   //Step 100 On EXIT - Store Identification
   IF #Step100ExitPls THEN
       #VD_Identification := #IO_VIDS.VEMData.Identification;
   END_IF;

   (******************************************************************************)
   (* Step 100 to 300                                                            *)
   (******************************************************************************)

   //Step 100 to 300
   IF #Step100To300Cond THEN
       #StepNbr := 300;
       #Step300EntryPls := TRUE;
   ELSE
       #Step300EntryPls := FALSE;
   END_IF;

   //Step 100 to 300 - Condition
   #Step100To300Cond :=
   #StepNbr = 100 AND
   #IO_VIDS.VEMData.CommandCode = 1001 AND
   #Status > 0 AND
   (#IO_VIDS.IDType = 0 AND #IO_VIDS.VEMData.Identification <> 0 OR #IO_VIDS.IDType > 0 AND #IO_VIDS.VEMData.CarrierID <> 0) AND
   NOT #NewData;

   (******************************************************************************)
   (* Step 200 - Send data                                                       *)
   (******************************************************************************)

   //Step 200 - On Entry - Check VEM data
   #DataValidSnd := #Step200EntryPls AND #IO_VIDS.VEMData.CommandCode <> 0;

   //Step 200 - On Entry - Check VEM data - Error
   IF #Step200EntryPls AND NOT #DataValidSnd THEN
       #Status := #STATUS_MINUS_006;
   END_IF;

   //Step 200 On Entry - VDCommLocalSndDB - Send VEM data TO virtual device
   IF #Step200EntryPls AND #Status > 0 THEN
       #SerializePos := 0;
       #RetVal:=Serialize(SRC_VARIABLE:=#IO_VIDS.VEMData, DEST_ARRAY=>#VEMDataSndArray, POS:=#SerializePos);
       #RetVal:=BLKMOV(SRCBLK := #VEMDataSndArray, DSTBLK => #ptrVEMDataVDCommLocalSnd);
       #RetVal:=BLKMOV(SRCBLK := #IO_VIDS.SpecificDataInit, DSTBLK => #ptrSpecDataVDCommLocalSnd);
       #CmdCodeSent := #IO_VIDS.VEMData.CommandCode;
   END_IF;

   //Step 200 on Active - Step Timer - Start
   #_Step200Tmr(I_StartTimer := #StepNbr = 200,
                I_HoldTimer := FALSE,
                I_MaxTimerValue := 15000,
                O_TimerResult => #Step200TmrElapsed,
                O_TimerValue => #Step200TmrAct);

   //Step 200 On Active - Step Timer - Error overtime
   IF #Step200TmrElapsed THEN
       #Status := #STATUS_MINUS_003;
   END_IF;

   //Step 200 On Active - Step Timer - Memorize maximum
   IF #Step200TmrAct > #Step200TmrActMax THEN
       #Step200TmrActMax := #Step200TmrAct;
   END_IF;

   //Step 200 On Active - Send TO VD
   #SendToVD := #StepNbr = 200 AND #Status>0;

   (******************************************************************************)
   (* Step 200 to 300                                                            *)
   (******************************************************************************)

   //Step 200 to 300
   IF #Step200To300Cond THEN
       #StepNbr := 300;
       #Step200ExitPls := TRUE;
   ELSE
       #Step200ExitPls := FALSE;
   END_IF;

   //Step 200 to 300 - Condition
   #Step200To300Cond := #StepNbr = 200 AND #SendFinished AND #Status > 0;

   (******************************************************************************)
   (* Step 300                                                                   *)
   (******************************************************************************)

   //Step 300 On Entry - VDCommLocalRcvDB - Create pointer TO VEM data
   #ptrVEMDataVDCommLocalRcvStruct.ID := #POINTER_SYNTAX_ID;
   #ptrVEMDataVDCommLocalRcvStruct.DataType := #DATA_TYPE_BYTE;
   #ptrVEMDataVDCommLocalRcvStruct.ReplicationFactor := 256;
   #ptrVEMDataVDCommLocalRcvStruct.DbNbr := UINT_TO_WORD(DB_ANY_TO_UINT(#C_VDCommLocalRcvDB));
   #ptrVEMDataVDCommLocalRcvStruct.CrossAreaPointer := SHL(IN := #VDCOM_VEM_DATA_OFFSET, N := 3) OR #AREA_IDENTIFIER; //Offset 10

   //Step 300 On Entry - VDCommLocalRcvDB - Create pointer TO Specific data
   #ptrSpecDataVDCommLocalRcvStruct.ID := #POINTER_SYNTAX_ID;
   #ptrSpecDataVDCommLocalRcvStruct.DataType := #DATA_TYPE_BYTE;
   #ptrSpecDataVDCommLocalRcvStruct.ReplicationFactor := 2048;
   #ptrSpecDataVDCommLocalRcvStruct.DbNbr := UINT_TO_WORD(DB_ANY_TO_UINT(#C_VDCommLocalRcvDB));
   #ptrSpecDataVDCommLocalRcvStruct.CrossAreaPointer := SHL(IN := #VDCOM_SPEC_DATA_OFFSET, N := 3) OR #AREA_IDENTIFIER; //Offset 10

   //Step 300 On Active - Receive data from virtual device
   IF #StepNbr = 300 AND #NewData THEN

       //Copy received data to VEM data receive structure
       #RetVal := BLKMOV(SRCBLK := #ptrVEMDataVDCommLocalRcv, DSTBLK => #VEMDataRcvArray);
       #DeserializePos := 0;
       #RetVal := Deserialize(SRC_ARRAY := #VEMDataRcvArray, DEST_VARIABLE => #VEMDataRcv, POS := #DeserializePos);

       //Received command code
       #CmdCodeRcvd := #VEMDataRcv.CommandCode;

       //Check error code
       IF #VEMDataRcv.ErrorCode < 0 THEN
           #Status := DINT_TO_INT(#VEMDataRcv.ErrorCode);
           //Data not Valid signal
           #VEMDataNotValid := TRUE;
       ELSE
           //Check data
           #DataValidRcv := NOT #IO_VIDS.GetVEMDataByRFID.Running AND
           #VEMDataRcv.CommandCode = #IO_VIDS.VEMData.CommandCode;

           #DataValidRcvGetVEMDataByRFID := #IO_VIDS.GetVEMDataByRFID.Running AND
           ((#VEMDataRcv.IdType = 0 AND #VEMDataRcv.Identification <> 0) OR (#VEMDataRcv.IdType <> 0 AND #VEMDataRcv.CarrierID <> 0));

           IF #DataValidRcv OR #DataValidRcvGetVEMDataByRFID THEN

               //Status 001 : Success
               #Status := #STATUS_001;

               //Copy all data
               #DeserializePos := 0;
               #RetVal := Deserialize(SRC_ARRAY := #VEMDataRcvArray, DEST_VARIABLE => #IO_VIDS.VEMData, POS := #DeserializePos);
               #RetVal := BLKMOV(SRCBLK := #ptrSpecDataVDCommLocalRcv, DSTBLK => #IO_SpecificData);
               #DeserializePos := 0;
               #RetVal := Deserialize(SRC_ARRAY := #VEMDataRcvArray, DEST_VARIABLE => #IO_VEMData, POS := #DeserializePos);
               #DeserializePos := 0;
               #RetVal := Deserialize(SRC_ARRAY := #VEMDataRcvArray, DEST_VARIABLE => #IO_VEMDataChange, POS := #DeserializePos);

               //Data Valid signal
               #VEMDataValid := TRUE;

           ELSE
               #VEMDataNotValid := TRUE;
               #Status := #STATUS_MINUS_005;
           END_IF;
       END_IF;
   END_IF;

   //Step 300 on Active - Step Timer - Start
   #_Step300Tmr(I_StartTimer := #StepNbr = 300,
                I_HoldTimer := FALSE,
                I_MaxTimerValue := 15000,
                O_TimerResult => #Step300TmrElapsed,
                O_TimerValue => #Step300TmrAct);

   //Step 300 On Active - Step Timer - Error overtime
   IF #Step300TmrElapsed THEN
       #Status := #STATUS_MINUS_009;
   END_IF;

   //Step 300 On Active - Step Timer - Memorize maximum
   IF #Step300TmrAct > #Step300TmrActMax THEN
       #Step300TmrActMax := #Step300TmrAct;
   END_IF;

   (******************************************************************************)
   (* Step 300 to 400                                                            *)
   (******************************************************************************)

   //Step 300 to 400
   IF #Step300To400Cond THEN
       #StepNbr := 400;
       #Step300ExitPls := TRUE;
   ELSE
       #Step300ExitPls := FALSE;
   END_IF;

   //Step 300 TO 400 - Condition
   #Step300To400Cond := #StepNbr = 300 AND #Status = 1;

   (******************************************************************************)
   (* Step XXX to 400                                                            *)
   (******************************************************************************)

   //Step XXX TO 400
   IF #StepNbr > 0 AND #Status < 0 THEN
       #VEMDataNotValid := TRUE;
       #StepNbr := 400;
   END_IF;

   (******************************************************************************)
   (* Step 400 to 0                                                              *)
   (******************************************************************************)

   //Step 400 to 0
   IF #Step400To0Cond THEN
       #StepNbr := 0;
       #Step400ExitPls := TRUE;
   ELSE
       #Step400ExitPls := FALSE;
   END_IF;

   //Step 400 TO 0 - Condition
   #Step400To0Cond := #StepNbr = 400;

   (******************************************************************************)
   (* Step 400 - Finish & Final Status                                           *)
   (******************************************************************************)

   //Step 400 On active - Finish & Final Status
   IF #StepNbr = 400 THEN

       IF #IO_VIDS.GetVEMData.Running THEN
           #IO_VIDS.GetVEMData.Running := FALSE;
           #IO_VIDS.GetVEMData.Status := #Status;
           #IO_VIDS.GetVEMData.Finished := TRUE;
       ELSIF #IO_VIDS.ChangeData.Running THEN
           #IO_VIDS.ChangeData.Running := FALSE;
           #IO_VIDS.ChangeData.Status := #Status;
           #IO_VIDS.ChangeData.Finished := TRUE;
       ELSIF #IO_VIDS.InitTag.Running THEN
           #IO_VIDS.InitTag.Running := FALSE;
           #IO_VIDS.InitTag.Status := #Status;
           #IO_VIDS.InitTag.Finished := TRUE;
       ELSIF #IO_VIDS.GetVEMDataByRFID.Running THEN
           #IO_VIDS.GetVEMDataByRFID.Running := FALSE;
           #IO_VIDS.GetVEMDataByRFID.Status := #Status;
           #IO_VIDS.GetVEMDataByRFID.Finished := TRUE;
       ELSIF #IO_VIDS.ReplaceTag.Running THEN
           #IO_VIDS.ReplaceTag.Running := FALSE;
           #IO_VIDS.ReplaceTag.Status := #Status;
           #IO_VIDS.ReplaceTag.Finished := TRUE;
       ELSIF #IO_VIDS.Track.Running THEN
           #IO_VIDS.Track.Running := FALSE;
           #IO_VIDS.Track.Status := #Status;
           #IO_VIDS.Track.Finished := TRUE;
       ELSIF #IO_VIDS.Confirm.Running THEN
           #IO_VIDS.Confirm.Running := FALSE;
           #IO_VIDS.Confirm.Status := #Status;
           #IO_VIDS.Confirm.Finished := TRUE;
       ELSIF #IO_VIDS.Couple.Running THEN
           #IO_VIDS.Couple.Running := FALSE;
           #IO_VIDS.Couple.Status := #Status;
           #IO_VIDS.Couple.Finished := TRUE;
       ELSIF #IO_VIDS.DeCouple.Running THEN
           #IO_VIDS.DeCouple.Running := FALSE;
           #IO_VIDS.DeCouple.Status := #Status;
           #IO_VIDS.DeCouple.Finished := TRUE;
       ELSIF #IO_VIDS.GetNextID.Running THEN
           #IO_VIDS.GetNextID.Running := FALSE;
           #IO_VIDS.GetNextID.Status := #Status;
           #IO_VIDS.GetNextID.Finished := TRUE;
       ELSIF #IO_VIDS.GetSpecData.Running THEN
           #IO_VIDS.GetSpecData.Running := FALSE;
           #IO_VIDS.GetSpecData.Status := #Status;
           #IO_VIDS.GetSpecData.Finished := TRUE;
       ELSIF #IO_VIDS.PutSpecData.Running THEN
           #IO_VIDS.PutSpecData.Running := FALSE;
           #IO_VIDS.PutSpecData.Status := #Status;
           #IO_VIDS.PutSpecData.Finished := TRUE;
       END_IF;

   ELSE

       #IO_VIDS.GetVEMData.Finished := FALSE;
       #IO_VIDS.ChangeData.Finished := FALSE;
       #IO_VIDS.InitTag.Finished := FALSE;
       #IO_VIDS.GetVEMDataByRFID.Finished := FALSE;
       #IO_VIDS.ReplaceTag.Finished := FALSE;
       #IO_VIDS.Track.Finished := FALSE;
       #IO_VIDS.Confirm.Finished := FALSE;
       #IO_VIDS.Couple.Finished := FALSE;
       #IO_VIDS.DeCouple.Finished := FALSE;
       #IO_VIDS.GetNextID.Finished := FALSE;
       #IO_VIDS.GetSpecData.Finished := FALSE;
       #IO_VIDS.PutSpecData.Finished := FALSE;

   END_IF;

   (******************************************************************************)
   (* CPU1500 - VDComSubSystem                                                   *)
   (******************************************************************************)

   //Reset NewData
   #ResetNewData:=#NewData;

   #MessageLength := DWORD_TO_WORD(#IO_VIDS.VEMData.SpecificDataLength+266);

   #"_LVDComSubSystemS7-1500"(I_CommunicationReset:=#ResetAllRequests,
                              I_SendRequest:=#SendToVD,
                              I_ResetNewData:=#ResetNewData,
                              I_MasterNewMessage:=#IO_VDComm.NewMessageVD,
                              I_MasterSendFinished:=#IO_VDComm.MessageSendDoneVD,
                              I_VDCommRecvDB:=#C_VDCommMasterRcvDB,
                              I_VDCommSendDB:=#C_VDCommMasterSndDB,
                              C_LocalRecvDB:=#C_VDCommLocalRcvDB,
                              C_LocalSendDB:=#C_VDCommLocalSndDB,
                              C_MessType:=20562,
                              C_SubSystem:=#C_SubSystem,
                              C_SendMessLen:=#MessageLength,
                              O_SendFinished=>#SendFinished,
                              O_NewData=>#NewData,
                              IO_MasterSendReq:=#IO_VDComm.MasterSendReq,
                              IO_MasterAckReq:=#IO_VDComm.MasterAckReq,
                              IO_SubSystemDBNr:=#IO_VDComm.VDCommSendDBNr,
                              IO_VDCommSendDB:=#IO_VDComm.VDCommSendDB);


   (******************************************************************************)
   (* Common signals to all submodules                                           *)
   (******************************************************************************)

   //Common signals to all submodules
   #IO_VIDS.PartPres := #PartPres;
   #IO_VIDS.IDType := #C_IDType;
   #IO_VIDS.VEMDataValid := #VEMDataValid;
   #IO_VIDS.VEMDataNotValid := #VEMDataNotValid;
   #IO_VIDS.CmdCodeRcvd := #CmdCodeRcvd;
   #IO_VIDS.CmdCodeSent := #CmdCodeSent;

   (******************************************************************************)
   (* Outputs                                                                    *)
   (******************************************************************************)

   IF #SECTION_OUTPUTS THEN

       #O_GetVEMDataBusy := #BusyGetVEMData;
       #O_Status := #Status;
       #O_Alarm := #Status < 0;
       #O_VEMDataValid := #VEMDataValid;
       #O_VEMDataNotValid := #VEMDataNotValid;

   END_IF;

   (******************************************************************************)
   (* HMI                                                                        *)
   (******************************************************************************)

   IF #SECTION_HMI THEN

       //Decode - BodyType matrix - Car type
       #CarTypeBody := DINT_TO_INT(DWORD_TO_DINT(#IO_VEMData.BodyTypeMatrix) / 100000);

       //Decode - BodyType matrix - Steering
       #SteeringBody := DINT_TO_INT((DWORD_TO_DINT(#IO_VEMData.BodyTypeMatrix) / 100000) MOD 10);

       //Decode - Variant - Car type - First digit
       #CarTypeArray[1] := (CHAR_TO_INT(#IO_VEMData.Variant[1]) - 48) * 100;
       #CarTypeArray[2] := (CHAR_TO_INT(#IO_VEMData.Variant[2]) - 48) * 10;
       #CarTypeArray[3] := (CHAR_TO_INT(#IO_VEMData.Variant[3]) - 48);

       //Decode - Variant - Car type - Summary digits
       #CarTypeVariant := #CarTypeArray[1] + #CarTypeArray[2] + #CarTypeArray[3];

       //Decode - Variant - Steering
       #SteeringVariant := #IO_VEMData.Variant[10];

       //HMI - Message - Part Present - Visible
       IF #IO_VIDS.PartPres THEN
           #H_Master.H_msgPartPresAnim := #VISIBLE;
       ELSE
           #H_Master.H_msgPartPresAnim := #OFF;
       END_IF;

       //HMI - Message - VEM Data Valid - Visible
       IF #VEMDataValid THEN
           #H_Master.H_msgVEMDataValidAnim := #VISIBLE;
       ELSE
           #H_Master.H_msgVEMDataValidAnim := #OFF;
       END_IF;

       //HMI - Message - VEM Data not Valid - Visible
       IF #VEMDataNotValid THEN
           #H_Master.H_msgVEMDataNotValidAnim := #VISIBLE;
       ELSE
           #H_Master.H_msgVEMDataNotValidAnim := #OFF;
       END_IF;

       //HMI - Value - Command code sent
       #H_Master.H_txtCommandCodeSent := #CmdCodeSent;

       //HMI - Value - Command code received
       #H_Master.H_txtCommandCodeRcvd := #CmdCodeRcvd;

       (******************************************************************************)
       (* HMI - Vehicle types                                                        *)
       (******************************************************************************)

       //HMI - Message - Body VEM data
       IF #C_IDType = 0 THEN
           #H_Master.H_msgVEMDataBody := 1;
       ELSE
           #H_Master.H_msgVEMDataBody := 0;
       END_IF;

       //HMI - Message - Carrier VEM data
       IF #C_IDType = 0 THEN
           #H_Master.H_msgVEMDataCarrier := 1;
       ELSE
           #H_Master.H_msgVEMDataCarrier := 0;
       END_IF;

       #H_Master.H_txtIdentification := #IO_VEMData.Identification;                    //HMI - Value - TagID
       #H_Master.H_txtBodyID := #IO_VEMData.BodyID;                                    //HMI - Value - BodyID
       #H_Master.H_txtCarrierID := #IO_VEMData.CarrierID;                              //HMI - Value - CarrierID
       #H_Master.H_txtBodyTypeMatrix := #IO_VEMData.BodyTypeMatrix;                    //HMI - Value - Bodytype matrix
       #H_Master.H_txtRouting := #IO_VEMData.Routing;                                  //HMI - Value - Routing
       #H_Master.H_txtCarrierDestination := #IO_VEMData.Destination;                   //HMI - Value - Carrier Destination
       #H_Master.H_txtWorkUntil := #IO_VEMData.WorkUntil;                              //HMI - Value - Work UNTIL Station
       #H_Master.H_txtWorkAfter := #IO_VEMData.BegWorkAfter;                           //HMI - Value - Start Work After Station
       #H_Master.H_txtBodyCargoStatus := #IO_VEMData.BodyCargoStatus ;                 //HMI - Value - Body Cargo Status
       #H_Master.H_txtCarrierCargoStatus := #IO_VEMData.CarrierCargoStatus;            //HMI - Value - Carrier Cargo Status
       #H_Master.H_txtEquipmentWork := #IO_VEMData.EquipmentWork;                      //HMI - Value - Equipment Work
       #H_Master.H_txtAvailabilityStatus := #IO_VEMData.AvailabilityStatus;            //HMI - Value - Availability Status
       #H_Master.H_txtModelYear := #IO_VEMData.ModelYear;                              //HMI - Value - ModelYear
       #H_Master.H_txtPreSerieInfo := #IO_VEMData.PreSerieInfo;                        //HMI - Value - Preseries Info
       #H_Master.H_txtWorkStatus := #IO_VEMData.WorkStatus;                            //HMI - Value - Work Status
       #H_Master.H_txtBodyType1 := #IO_VEMData.BodyType1;                              //HMI - Value - Bodytype 1
       #H_Master.H_txtBodyType2 := #IO_VEMData.BodyType2;                              //HMI - Value - Bodytype 2
       #H_Master.H_txtRobotProgramNumber := #IO_VEMData.RobotProgramNumber;            //HMI - Value - Robot Program Number
       #H_Master.H_txtPLCProgramNbr := #H_Master.H_txtPLCProgramNbr;                   //HMI - Value - PLC Program Number
       #H_Master.H_txtEquipmentWorkDone := #IO_VEMData.EquipmentWorkDone;              //HMI - Value - Equipment Work Done
       #H_Master.H_txtSequenceNumber := #IO_VEMData.SequenceNumber;                    //HMI - Value - Sequence Number
       #H_Master.H_txtBufferIn := #IO_VEMData.BufferIn;                                //HMI - Value - BufferIn
       #H_Master.H_txtBufferOut := #IO_VEMData.BufferOut;                              //HMI - Value - BufferOut
       #H_Master.H_txtCarrierType := #IO_VEMData.CarrierType;                          //HMI - Value - Carrier Type
       #H_Master.H_txtCarrierLapCounter := #IO_VEMData.CarrierLapCounter;              //HMI - Value - Carrier Lap Counter
       #H_Master.H_txtCarrierIDUBFlow := #IO_VEMData.CarrierIDUBFlow;                  //HMI - Value - Carrier ID UB Flow
       #H_Master.H_txtCarrierBodyType := #IO_VEMData.CarrierBodyType;                  //HMI - Value - Carrier Bodytype
       #H_Master.H_txtAddQualityItemEquipment := #IO_VEMData.AddQualityItemEquipment;  //HMI - Value - Add Quality Item Equipment
       #H_Master.H_txtChkQualityItemEquipment := #IO_VEMData.CheckQualityItemEquipment;//HMI - Value - Check Quality Item Equipment
       #H_Master.H_txtCarrierMaxCycleCounter := #IO_VEMData.CarrierMaxCycleCount;      //HMI - Value - CarrMaxCycleCntr    
       #H_Master.H_txtSurfacerColour := #IO_VEMData.SurfacerColour;                    //HMI - Value - SurfacerColour
       #H_Master.H_txtTopCoatColour := #IO_VEMData.TopCoatColour;                      //HMI - Value - TopCoatColour
       #H_Master.H_txtClearCoatColour := #IO_VEMData.ClearCoatColour;                  //HMI - Value - ClearCoatColour
       #H_Master.H_txtPopType := #IO_VEMData.PopType;                                  //HMI - Value - PopType
       #H_Master.H_txtPopId := #IO_VEMData.PopID;                                      //HMI - Value - PopId
       #H_Master.H_txtPopIdSuffix := #IO_VEMData.PopIDSuffix;                          //HMI - Value - PopId

       //HMI - Value - Variant
       FOR #i := 1 TO 8 DO
           #H_Master.H_txtVariant[#i] := #IO_VEMData.Variant[#i];
       END_FOR;

       //HMI - Value - VIN number
       FOR #i := 1 TO 20 DO
           #H_Master.H_txtVinNumber[#i - 1] := #IO_VEMData.VinNumber[#i];
       END_FOR;

       #H_Master.H_txtMixNumber := #IO_VEMData.MixNumber;                          //HMI - Value - Mixnumber
       #H_Master.H_txtIDType := #IO_VEMData.IdType;                                // HMI - Value - ID Type

       //HMI - Message - Running 
       #H_Master.H_msgFunctionNbrAnim := 0;                //Reset animation before we begin

       //HMI - Message - Running - Get VEM Data
       IF #IO_VIDS.GetVEMData.Running THEN
           #H_Master.H_msgFunctionNbrAnim := 1;
       END_IF;

       //HMI - Message - Running - Change VEM Data
       IF #IO_VIDS.ChangeData.Running THEN
           #H_Master.H_msgFunctionNbrAnim := 2;
       END_IF;

       //HMI - Message - Running - Init
       IF #IO_VIDS.InitTag.Running THEN
           #H_Master.H_msgFunctionNbrAnim := 3;
       END_IF;

       //HMI - Message - Running - Get VEM Data by RFID
       IF #IO_VIDS.GetVEMDataByRFID.Running THEN
           #H_Master.H_msgFunctionNbrAnim := 4;
       END_IF;

       //HMI - Message - Running - Replace tag
       IF #IO_VIDS.ReplaceTag.Running THEN
           #H_Master.H_msgFunctionNbrAnim := 5;
       END_IF;

       //HMI - Message - Running - Track
       IF #IO_VIDS.Track.Running THEN
           #H_Master.H_msgFunctionNbrAnim := 6;
       END_IF;

       //HMI - Message - Running - Confirm
       IF #IO_VIDS.Confirm.Running THEN
           #H_Master.H_msgFunctionNbrAnim := 7;
       END_IF;

       //HMI - Message - Running - Couple
       IF #IO_VIDS.Couple.Running THEN
           #H_Master.H_msgFunctionNbrAnim := 8;
       END_IF;

       //HMI - Message - Running - Decouple
       IF #IO_VIDS.DeCouple.Running THEN
           #H_Master.H_msgFunctionNbrAnim := 9;
       END_IF;

       //HMI - Message - Running - Get Next ID
       IF #IO_VIDS.GetNextID.Running THEN
           #H_Master.H_msgFunctionNbrAnim := 10;
       END_IF;

       //HMI - Message - Running - Get Specific Data
       IF #IO_VIDS.GetSpecData.Running THEN
           #H_Master.H_msgFunctionNbrAnim := 11;
       END_IF;

       //HMI - Message - Running - Put Specific Data
       IF #IO_VIDS.PutSpecData.Running THEN
           #H_Master.H_msgFunctionNbrAnim := 12;
       END_IF;

       #H_Master.H_msgStepNbrAnim := INT_TO_WORD(#StepNbr);             //HMI - Message - StepNumber

       //Update step timers
       IF #StepNbr = 100 THEN
           #H_Master.H_txtStep100TmrMax := DINT_TO_INT(#Step100TmrAct);  //HMI - Step 100 Timer
       ELSIF #StepNbr = 200 THEN
           #H_Master.H_txtStep200TmrMax := DINT_TO_INT(#Step200TmrAct);  //HMI - Step 200 Timer
       ELSIF #StepNbr = 300 THEN
           #H_Master.H_txtStep300TmrMax := DINT_TO_INT(#Step300TmrAct);  //HMI - Step 300 Timer
       END_IF;

       //Reset Step timers
       IF #H_Master.H_btnResetStepTimers <> 0 THEN
           #H_Master.H_txtStep100TmrMax := 0;
           #H_Master.H_txtStep200TmrMax := 0;
           #H_Master.H_txtStep300TmrMax := 0;
       END_IF;

       #H_Master.H_msgStatus := #Status;                   //HMI - Status

       // HMI - Icon animation
       "LIAnimDWord"(I_SetPos := FALSE,
                     I_ResetPos := FALSE,
                     I_Active := #Status > 1,
                     I_Visible := FALSE,
                     I_OutOfUse := FALSE,
                     I_IntlkSet := FALSE,
                     I_IntlkReset := FALSE,
                     I_IntlkSetAlm := FALSE,
                     I_IntlkResetAlm := FALSE,
                     I_ManualMode := FALSE,
                     I_FncSelInHMI := FALSE,
                     I_AnySelected := FALSE,
                     I_AlarmA := FALSE,
                     I_AlarmB := FALSE,
                     I_AlarmC := #Status < 0,
                     I_AlarmD := FALSE,
                     I_SafetyOk := FALSE,
                     I_Service:="TRUE",
                     I_Spare1:="FALSE",
                     I_Spare2:="FALSE",
                     I_Spare3:="FALSE",
                     I_Spare4:="FALSE",
                     I_Spare5:="FALSE",
                     I_Spare6:="FALSE",
                     I_Spare7:="FALSE",
                     I_Spare8:="FALSE",
                     I_Spare9:="FALSE",
                     I_Spare10:="FALSE",
                     I_Spare11:="FALSE",
                     I_Spare12:="FALSE",
                     I_Spare13:="FALSE",
                     I_Spare14:="FALSE",
                     H_IAnim => #H_HMI.H_IAnim);

   (******************************************************************************)
   (* HMI - Reset buttons                                                        *)
   (******************************************************************************)

       #H_Master.H_btnResetStepTimers := #OFF;
       #H_Master.H_btnGetVEMDataByTagID := #OFF;
       #H_Master.H_btnGetVEMDataByBodyID := #OFF;
       #H_Master.H_btnGetVEMDataByCarrierID := #OFF;
       #H_Master.H_btnGetVEMDataByMixNbr := #OFF;

   END_IF;

   (******************************************************************************)
   (* Alarm                                                                      *)
   (******************************************************************************)

   #Alarm := (#Status < 0);

   "LAlarmSummary"(I_AlarmA := "FALSE",
                   I_AlarmB := "FALSE",
                   I_AlarmC := #Alarm,
                   I_AlarmD := "FALSE",
                   I_AlarmABCondition := "FALSE",
                   IO_Alarm := #IO_Alarm,
                   C_UpperLevelHW := "FALSE",
                   C_UpperLevelSafety := "FALSE",
                   C_Safety := "FALSE",
                   C_Mechanic := "FALSE",
                   C_Transport := "FALSE",
                   C_Feature1 := "FALSE",
                   C_Feature2 := "FALSE",
                   C_Feature3 := "FALSE");
END_FUNCTION_BLOCK

FUNCTION_BLOCK "LVDComSubSystemS7-1500"   // FB2215, FBD
TITLE = VDComSubSystemS7-1500
{ S7_Optimized_Access := 'FALSE' }
AUTHOR : VCC
FAMILY : Communic
VERSION : 0.1
// =============================================================================
// This Module Extract Data From VDCom Send/Recv
// =============================================================================
// stored: AutoNumber false, IsIECCheckEnabled false, SetENOAutomatically False, UDAEnableTagReadback false
   VAR_INPUT
      I_CommunicationReset { ExternalAccessible := 'False'; ExternalVisible := 'False'; ExternalWritable := 'False'} : Bool;   // Reset communication by Application
      I_SendRequest { ExternalAccessible := 'False'; ExternalVisible := 'False'; ExternalWritable := 'False'} : Bool;   // Send Command by Application
      I_ResetNewData { ExternalAccessible := 'False'; ExternalVisible := 'False'; ExternalWritable := 'False'} : Bool;   // Trigger by Application to Reset output "NewData"
      I_MasterNewMessage { ExternalAccessible := 'False'; ExternalVisible := 'False'; ExternalWritable := 'False'} : Bool;   // Signal from MasterBlock to indicate new message.
      I_MasterSendFinished { ExternalAccessible := 'False'; ExternalVisible := 'False'; ExternalWritable := 'False'} : Bool;   // Acknowledge from MasterBlock that Send command has been performed
      I_VDCommRecvDB { ExternalAccessible := 'False'; ExternalVisible := 'False'; ExternalWritable := 'False'} : DB_ANY;   // VD communication system receive DB; Not to be used by Application
      I_VDCommSendDB { ExternalAccessible := 'False'; ExternalVisible := 'False'; ExternalWritable := 'False'} : DB_ANY;   // VD communication system send DB; Not to be used by Application
      C_LocalRecvDB { ExternalAccessible := 'False'; ExternalVisible := 'False'; ExternalWritable := 'False'} : DB_ANY;   // Local DB For Recv Data Used By The Application
      C_LocalSendDB { ExternalAccessible := 'False'; ExternalVisible := 'False'; ExternalWritable := 'False'} : DB_ANY;   // Local DB For Send Data Used By The Application
      C_MessType { ExternalAccessible := 'False'; ExternalVisible := 'False'; ExternalWritable := 'False'} : Int := 10;   // Identify Message
      C_SubSystem { ExternalAccessible := 'False'; ExternalVisible := 'False'; ExternalWritable := 'False'} : Int;   // Identify Subsystem
      C_SendMessLen { ExternalAccessible := 'False'; ExternalVisible := 'False'; ExternalWritable := 'False'} : Word;   // Number to identify the Length of the message
   END_VAR
   VAR_OUTPUT
      O_SendFinished { ExternalAccessible := 'False'; ExternalVisible := 'False'; ExternalWritable := 'False'} : Bool;   // Sending of Data is done; to Application
      O_NewData { ExternalAccessible := 'False'; ExternalVisible := 'False'; ExternalWritable := 'False'} : Bool;   // New data is available from SubSystem to Application
   END_VAR
   VAR_IN_OUT
      IO_MasterSendReq { ExternalAccessible := 'False'; ExternalVisible := 'False'; ExternalWritable := 'False'} : Bool;   // Request from the SubBlock to the MasterBlock to Send data
      IO_MasterAckReq { ExternalAccessible := 'False'; ExternalVisible := 'False'; ExternalWritable := 'False'} : Bool;   // Acknowledge to Master upon MessageType- and SubSystem Match
      IO_SubSystemDBNr { ExternalAccessible := 'False'; ExternalVisible := 'False'; ExternalWritable := 'False'} : Int;   // VD Communication Send DB number, Set by SubSystem
      IO_VDCommSendDB { ExternalAccessible := 'False'; ExternalVisible := 'False'; ExternalWritable := 'False'} : DB_ANY;   // VD Communication send DB
   END_VAR
   VAR DB_SPECIFIC
      ThisModuleActiveSend { ExternalAccessible := 'False'; ExternalVisible := 'False'; ExternalWritable := 'False'} : Bool;   // This module active for sending
      ThisModuleActiveRead { ExternalAccessible := 'False'; ExternalVisible := 'False'; ExternalWritable := 'False'} : Bool;   // This module active for Reading / acknowledge
      NewDataPulse { ExternalAccessible := 'False'; ExternalVisible := 'False'; ExternalWritable := 'False'} : Bool;   // Bit to create pulse on NewData
      NewData { ExternalAccessible := 'False'; ExternalVisible := 'False'; ExternalWritable := 'False'} : Bool;   // New Data
      NewDataAvailable { ExternalAccessible := 'False'; ExternalVisible := 'False'; ExternalWritable := 'False'} : Bool;   // New Data Available
      NewDataAvailablePulse { ExternalAccessible := 'False'; ExternalVisible := 'False'; ExternalWritable := 'False'} : Bool;   // New Data Available Pulse
      _RestartSend { ExternalAccessible := 'False'; ExternalVisible := 'False'; ExternalWritable := 'False'; S7_SetPoint := 'True'} : IEC_TIMER;
   END_VAR
   VAR_TEMP
      PtrRECV : Any;   // Pointer to the system receive DB
      PtrARECV : Any;   // Pointer to the Application receive DB
      RecvMessType : Int;   // Message type of the received data
      RecvSubSyst : Int;   // Subsystem target number
      RcvLength : Int;   // Length of received data
      RecvDBNbr : Int;   // Receive system DB Number
      SendDBNbr : Int;   // Send system DB Number
      LocalRecvDBNbr : Int;   // Receive DB Number Local by Application
      LocalSendDBNbr : Int;   // Send DB Number Local by Application
   END_VAR
   VAR_TEMP   // added for the SCL form of the ladder/FBD networks
      _w1 : Bool;
      _w2 : Bool;
   END_VAR
BEGIN

NETWORK
TITLE = **** 1 - Inputs **** Load DB
// Load DB numbers to local variables from the Receive and Send DB from - VD Master - VD Subsystem
// Read DB Number Recv
      OPN   #I_VDCommRecvDB;
      L     DBNO;
      T     #RecvDBNbr;

// Read DB Number Send
      OPN   #I_VDCommSendDB;
      L     DBNO;
      T     #SendDBNbr;

// DB Number from VD Sub system
      OPN   #C_LocalRecvDB;
      L     DBNO;
      T     #LocalRecvDBNbr;

// Read DB Number Send
      OPN   #C_LocalSendDB;
      L     DBNO;
      T     #LocalSendDBNbr;

REGION Network 2: **** 3.1 - Communication - Other Systems **** Reset Communications
   // Reset Communications
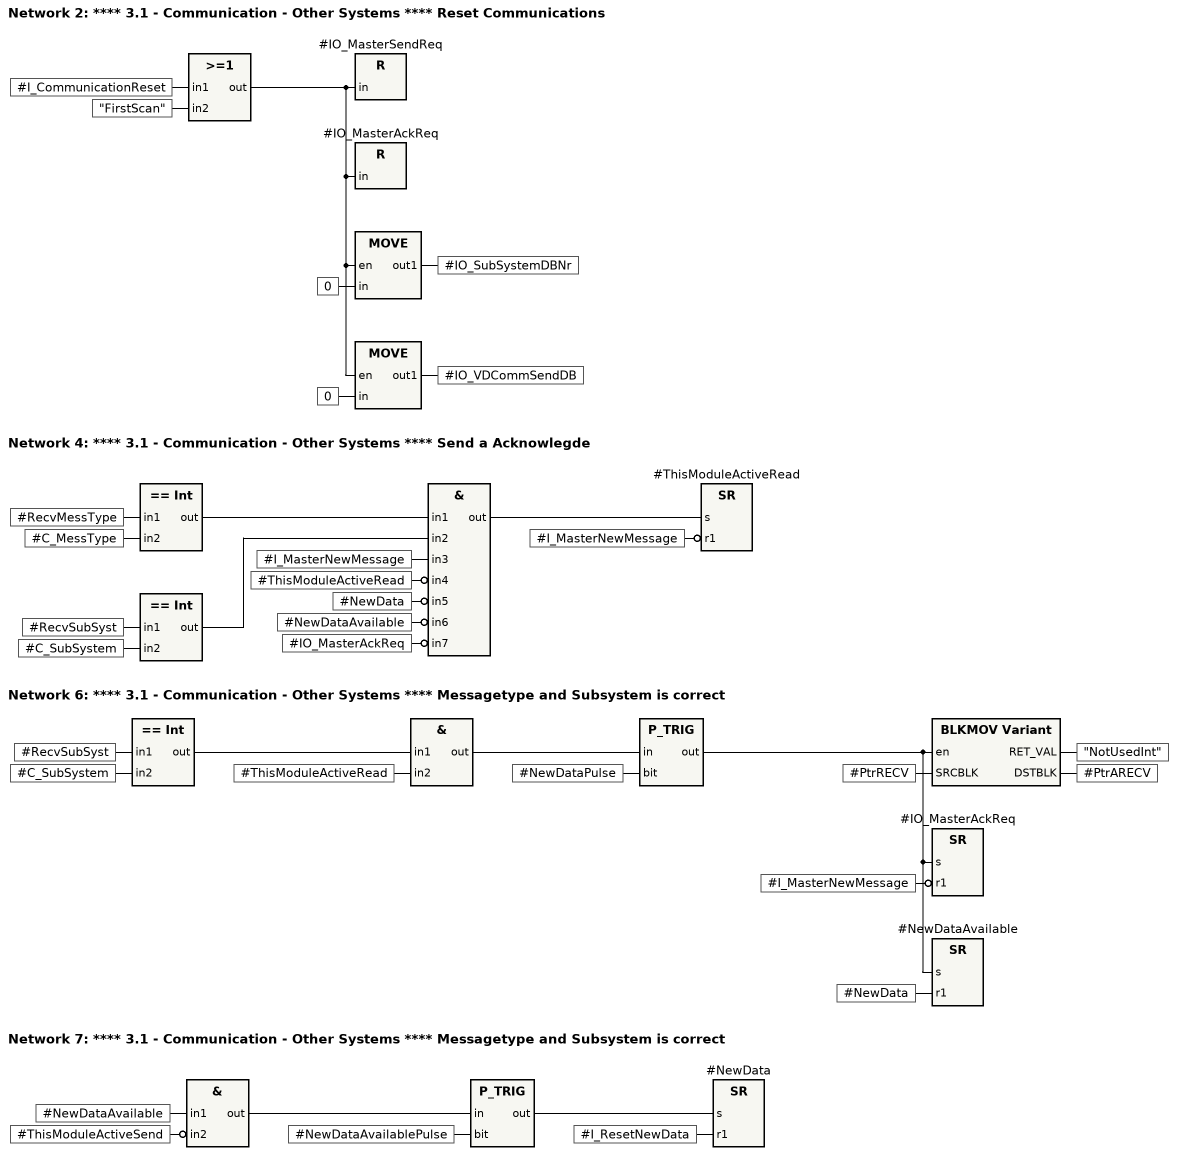
   IF #I_CommunicationReset OR "FirstScan" THEN
       #IO_MasterSendReq := FALSE;
       #IO_MasterAckReq := FALSE;
       #IO_SubSystemDBNr := 0;
       #IO_VDCommSendDB := 0;
   END_IF;
END_REGION

NETWORK
TITLE = **** 3.1 - Communication - Other Systems **** Header Information
// Copy Header information to local variables  Copy MessageType to local variable
      A     #ThisModuleActiveRead;
      JC    TMAR;
//OPN DB [ #RecvDBNbr] APa S7-1500
      OPN   #I_VDCommRecvDB;
      L     %DBW4;
      T     #RecvMessType;
//Copy SubSystemNbr to local variable
      L     %DBW6;
      T     #RecvSubSyst;
//Copy Lenth to local variable
      L     %DBW2;
      T     #RcvLength;
TMAR: NOP   0;

REGION Network 4: **** 3.1 - Communication - Other Systems **** Send a Acknowlegde
   // Send a Acknowlegde Request if Messagetype and Subsystem is correct
   IF (#RecvMessType = #C_MessType) AND (#RecvSubSyst = #C_SubSystem) AND #I_MasterNewMessage AND NOT #ThisModuleActiveRead AND NOT #NewData AND NOT #NewDataAvailable AND NOT #IO_MasterAckReq THEN
       #ThisModuleActiveRead := TRUE;   // SR flip-flop
   END_IF;
   IF NOT #I_MasterNewMessage THEN #ThisModuleActiveRead := FALSE; END_IF;
END_REGION

NETWORK
TITLE = **** 3.1 - Communication - Other Systems **** Configure DB
// Configure DB pointers
// APa Cleaning Warnings
      LAR1  P##PtrRECV;
      L     16#1002;
      T     LW [AR1, P#0.0];
      L     #RcvLength;
      T     LW [AR1, P#2.0];
      L     #RecvDBNbr;
      T     LW [AR1, P#4.0];
      L     0;
      SLD   3;
      OD    16#8400_0000;
      T     LD [AR1, P#6.0];

      LAR1  P##PtrARECV;
      L     16#1002;
      T     LW [AR1, P#0.0];
      L     #RcvLength;
      T     LW [AR1, P#2.0];
      L     #LocalRecvDBNbr;
      T     LW [AR1, P#4.0];
      L     0;
      SLD   3;
      OD    16#8400_0000;
      T     LD [AR1, P#6.0];
//      L     16#10                // S7  S7
//      T     %LB0
//      T     %LB10
//      L     16#02                // Data type to copy B#16#2 = Bytes
//      T     %LB1
//      T     %LB11
//      L     #RcvLength           //Length receiving data
//      T     %LW2
//      T     %LW12
//      L     #RecvDBNbr           // Receive DB Number
//      T     %LW4
//      L     #LocalRecvDBNbr      // Local Receive DB Number
//      T     %LW14
//      L     L#0                  //Offset in DB
//      SLD   3                    // Convert to pointer
//      T     %LD6
//      T     %LD16
//      L     16#84                // Memory area DB Memory area DB
//      T     %LB6
//      T     %LB16


REGION Network 6: **** 3.1 - Communication - Other Systems **** Messagetype and Subsystem is correct
   // New Data-flag if Messagetype and Subsystem is correct
   #_w1 := (#RecvSubSyst = #C_SubSystem) AND #ThisModuleActiveRead;
   #_w2 := #_w1 AND NOT #NewDataPulse;   // rising edge
   #NewDataPulse := #_w1;
   IF #_w2 THEN
       "NotUsedInt" := BLKMOV(SRCBLK := #PtrRECV, DSTBLK => #PtrARECV);
       #IO_MasterAckReq := TRUE;   // SR flip-flop
   END_IF;
   IF NOT #I_MasterNewMessage THEN #IO_MasterAckReq := FALSE; END_IF;
   IF #_w2 THEN
       #NewDataAvailable := TRUE;   // SR flip-flop
   END_IF;
   IF #NewData THEN #NewDataAvailable := FALSE; END_IF;
END_REGION

REGION Network 7: **** 3.1 - Communication - Other Systems **** Messagetype and Subsystem is correct
   // New Data-flag if Messagetype and Subsystem is correct
   #_w1 := #NewDataAvailable AND NOT #ThisModuleActiveSend;
   #_w2 := #_w1 AND NOT #NewDataAvailablePulse;   // rising edge
   #NewDataAvailablePulse := #_w1;
   IF #_w2 THEN
       #NewData := TRUE;   // SR flip-flop
   END_IF;
   IF #I_ResetNewData THEN #NewData := FALSE; END_IF;
END_REGION

NETWORK
TITLE = **** 3.1 - Communication - Other Systems **** Configure Header
// Configure Header for send data
//      OPN DB [ #LocalSendDBNbr] APa S7-1500
      OPN   #C_LocalSendDB;
      L     16#01;  //VD Version
      T     %DBB0;

      L     16#00;  //spare byte
      T     %DBB1;

//
      L     #C_SendMessLen;
      L     0;
      ==I;
      JC    Len1;
      L     #C_SendMessLen;
      JU    Len2;
Len1: L     DBLG;
Len2: T     %DBW2;

      L     #C_MessType;
      T     %DBW4;

      L     #C_SubSystem;
      T     %DBW6;


REGION Network 9: **** 3.1 - Communication - Other Systems **** This module is Active for Sending
   // This Module Active For Sending
   // - Check if no Request active (IO_MasterSendReq)
   // - Check if No DB Selected
   // - Check if Master does not send finished
   // - Send data Request from Application
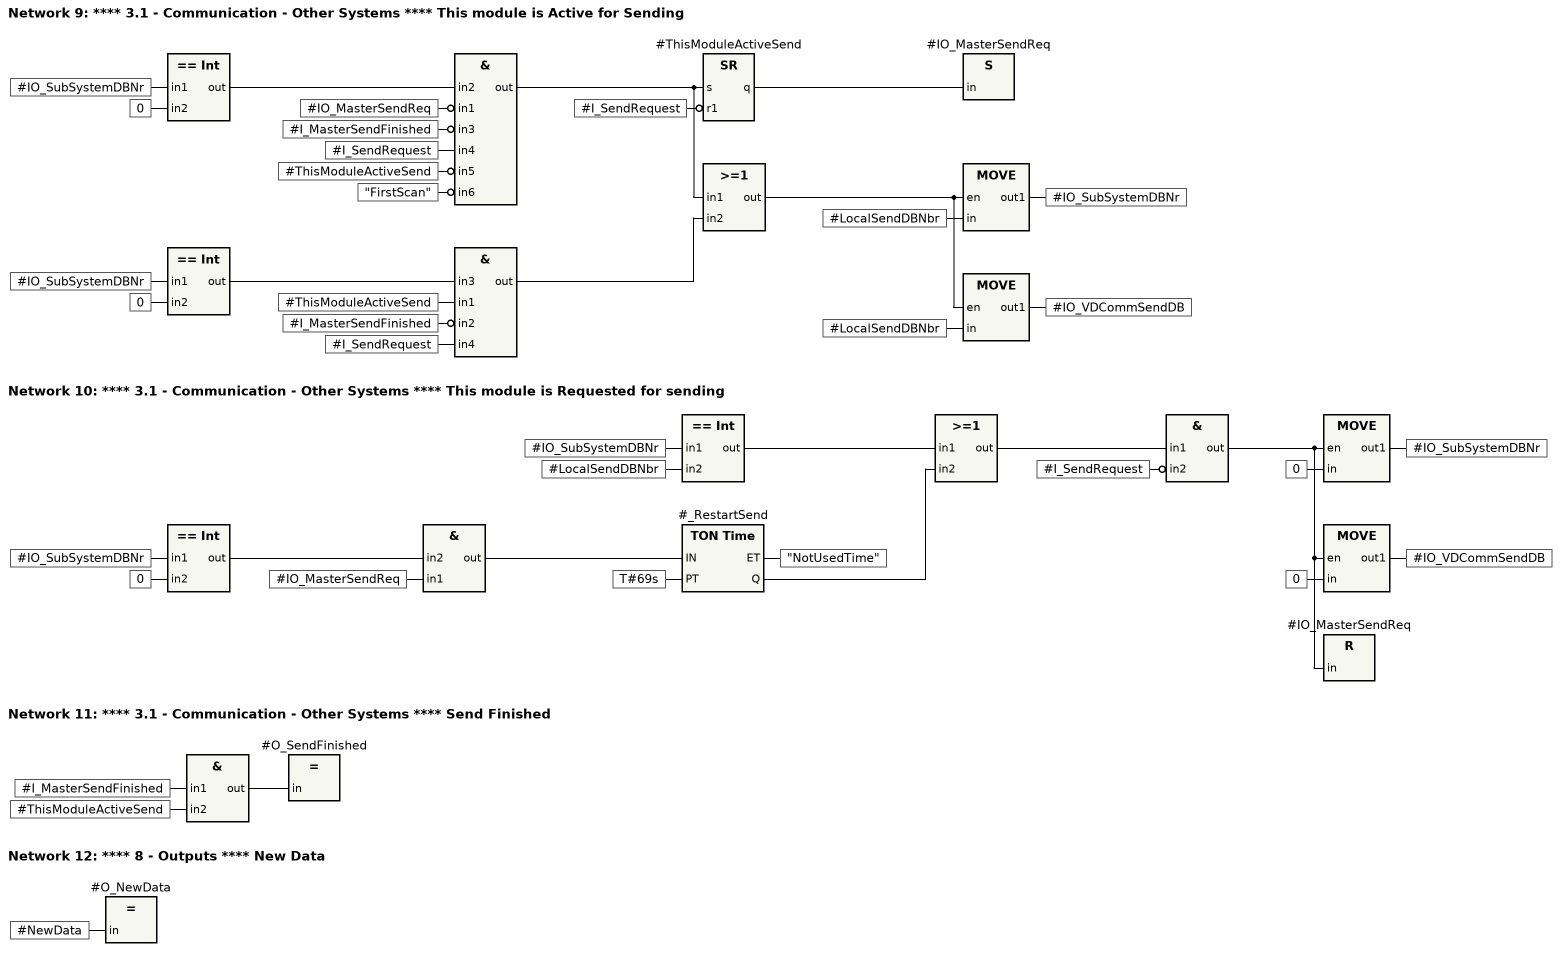
   #_w1 := (#IO_SubSystemDBNr = 0) AND NOT #IO_MasterSendReq AND NOT #I_MasterSendFinished AND #I_SendRequest AND NOT #ThisModuleActiveSend AND NOT "FirstScan";
   IF #_w1 THEN
       #ThisModuleActiveSend := TRUE;   // SR flip-flop
   END_IF;
   IF NOT #I_SendRequest THEN #ThisModuleActiveSend := FALSE; END_IF;
   IF #ThisModuleActiveSend THEN #IO_MasterSendReq := TRUE; END_IF;
   #_w2 := #_w1 OR ((#IO_SubSystemDBNr = 0) AND #ThisModuleActiveSend AND NOT #I_MasterSendFinished AND #I_SendRequest);
   IF #_w2 THEN
       #IO_SubSystemDBNr := #LocalSendDBNbr;
       #IO_VDCommSendDB := #LocalSendDBNbr;
   END_IF;
END_REGION

REGION Network 10: **** 3.1 - Communication - Other Systems **** This module is Requested for sending
   // This module is Requested for sending
   #_RestartSend.TON(IN := (#IO_SubSystemDBNr = 0) AND #IO_MasterSendReq, PT := T#69s, ET => "NotUsedTime");
   #_w1 := ((#IO_SubSystemDBNr = #LocalSendDBNbr) OR #_RestartSend.Q) AND NOT #I_SendRequest;
   IF #_w1 THEN
       #IO_SubSystemDBNr := 0;
       #IO_VDCommSendDB := 0;
       #IO_MasterSendReq := FALSE;
   END_IF;
END_REGION

REGION Network 11: **** 3.1 - Communication - Other Systems **** Send Finished
   // Send Finished
   #O_SendFinished := #I_MasterSendFinished AND #ThisModuleActiveSend;
END_REGION

REGION Network 12: **** 8 - Outputs **** New Data
   // New Data
   #O_NewData := #NewData;
END_REGION
END_FUNCTION_BLOCK

FUNCTION_BLOCK "LVIDSRFID"   // FB1203, SCL
{ S7_Optimized_Access := 'TRUE' }
VERSION : 0.1
// stored: AutoNumber false, IsIECCheckEnabled false, IsRetainMemResEnabled false, MemoryReserve 100, SetENOAutomatically False, UDAEnableTagReadback false
   VAR_INPUT
      I_OutOfUse { ExternalAccessible := 'False'; ExternalVisible := 'False'; ExternalWritable := 'False'} : Bool;   // Module out of use
      C_AntennaTriggOnTime { ExternalAccessible := 'False'; ExternalVisible := 'False'; ExternalWritable := 'False'} : DInt := 3000;   // Default 3s
      C_AntennaTriggOffTime { ExternalAccessible := 'False'; ExternalVisible := 'False'; ExternalWritable := 'False'} : DInt := 500;   // Default 500ms
      I_AntennaStatus { ExternalAccessible := 'False'; ExternalVisible := 'False'; ExternalWritable := 'False'} : Bool;   // Antenna status
      I_StartRead { ExternalAccessible := 'False'; ExternalVisible := 'False'; ExternalWritable := 'False'} : Bool;   // On edge, start tag read
      I_InitTagEn { ExternalAccessible := 'False'; ExternalVisible := 'False'; ExternalWritable := 'False'} : Bool := FALSE;   // Init tag enabled
      I_StartInitTag { ExternalAccessible := 'False'; ExternalVisible := 'False'; ExternalWritable := 'False'} : Bool;   // On edge, start initialisation
      I_BodyIDInitTag { ExternalAccessible := 'False'; ExternalVisible := 'False'; ExternalWritable := 'False'} : DWord;   // Body identifier for init function
      I_BodyType1InitTag { ExternalAccessible := 'False'; ExternalVisible := 'False'; ExternalWritable := 'False'} : DWord;   // BodyType1
      I_PopIDInitTag { ExternalAccessible := 'False'; ExternalVisible := 'False'; ExternalWritable := 'False'} : UDInt;   // Spare Data / PopID
      I_PopIDSuffixInitTag { ExternalAccessible := 'False'; ExternalVisible := 'False'; ExternalWritable := 'False'} : Char;   // PopID suffix
      I_PopTypeInitTag { ExternalAccessible := 'False'; ExternalVisible := 'False'; ExternalWritable := 'False'} : UDInt;   // Pop identifier
      I_ResetAlarm { ExternalAccessible := 'False'; ExternalVisible := 'False'; ExternalWritable := 'False'} : Bool;   // Reset alarm
   END_VAR
   VAR_OUTPUT
      O_AntennaTrigg { ExternalAccessible := 'False'; ExternalVisible := 'False'; ExternalWritable := 'False'} : Bool;   // to antenna - start read
      O_Busy { ExternalAccessible := 'False'; ExternalVisible := 'False'; ExternalWritable := 'False'} : Bool;   // Busy
      O_ReadOK { ExternalAccessible := 'False'; ExternalVisible := 'False'; ExternalWritable := 'False'} : Bool;   // RFID read OK
      O_ReadNOK { ExternalAccessible := 'False'; ExternalVisible := 'False'; ExternalWritable := 'False'} : Bool;   // RFID read NOK
      O_InitTagBusy { ExternalAccessible := 'False'; ExternalVisible := 'False'; ExternalWritable := 'False'} : Bool;   // Tag init busy
      O_InitTagOK { ExternalAccessible := 'False'; ExternalVisible := 'False'; ExternalWritable := 'False'} : Bool;   // Tag init OK
      O_InitTagNOK { ExternalAccessible := 'False'; ExternalVisible := 'False'; ExternalWritable := 'False'} : Bool;   // Tag init NOK
      O_ReplaceTagBusy { ExternalAccessible := 'False'; ExternalVisible := 'False'; ExternalWritable := 'False'} : Bool;
      O_ReplaceTagOK { ExternalAccessible := 'False'; ExternalVisible := 'False'; ExternalWritable := 'False'} : Bool;   // Replace tag - OK
      O_ReplaceTagNOK { ExternalAccessible := 'False'; ExternalVisible := 'False'; ExternalWritable := 'False'} : Bool;   // Replace tag - NOK
      O_Status { ExternalAccessible := 'False'; ExternalVisible := 'False'; ExternalWritable := 'False'} : Int;   // Status code
      O_Alarm { ExternalAccessible := 'False'; ExternalVisible := 'False'; ExternalWritable := 'False'} : Bool;   // Alarm C / Alarm
   END_VAR
   VAR_IN_OUT
      IO_VIDS : "VIDS";   // For internal use only
      IO_VEMData : "VEMData";   // From master module
      IO_Alarm : "Alarm";   // Alarm
      H_RFID : "H_LVIDSRFID";
      H_HMI : "H_HMI";
   END_VAR
   VAR
      i { ExternalAccessible := 'False'; ExternalVisible := 'False'; ExternalWritable := 'False'} : Int;   // Index
      Reset { ExternalAccessible := 'False'; ExternalVisible := 'False'; ExternalWritable := 'False'} : Bool;
      ReadOK { ExternalAccessible := 'False'; ExternalVisible := 'False'; ExternalWritable := 'False'} : Bool;
      ReadNOK { ExternalAccessible := 'False'; ExternalVisible := 'False'; ExternalWritable := 'False'} : Bool;
      InitTagOK { ExternalAccessible := 'False'; ExternalVisible := 'False'; ExternalWritable := 'False'} : Bool;
      InitTagNOK { ExternalAccessible := 'False'; ExternalVisible := 'False'; ExternalWritable := 'False'} : Bool;
      ReplaceTagOK { ExternalAccessible := 'False'; ExternalVisible := 'False'; ExternalWritable := 'False'} : Bool;
      ReplaceTagNOK { ExternalAccessible := 'False'; ExternalVisible := 'False'; ExternalWritable := 'False'} : Bool;
      StartReplaceTagMem { ExternalAccessible := 'False'; ExternalVisible := 'False'; ExternalWritable := 'False'} : Bool;
      StartInitMem { ExternalAccessible := 'False'; ExternalVisible := 'False'; ExternalWritable := 'False'} : Bool;
      btnForceReadEdg { ExternalAccessible := 'False'; ExternalVisible := 'False'; ExternalWritable := 'False'} : Bool;
      btnForceReadPls { ExternalAccessible := 'False'; ExternalVisible := 'False'; ExternalWritable := 'False'} : Bool;
      btnInitTagByBodyIdEdg { ExternalAccessible := 'False'; ExternalVisible := 'False'; ExternalWritable := 'False'} : Bool;
      btnInitTagByBodyIdPls { ExternalAccessible := 'False'; ExternalVisible := 'False'; ExternalWritable := 'False'} : Bool;
      btnInitTagByBodyType1Edg { ExternalAccessible := 'False'; ExternalVisible := 'False'; ExternalWritable := 'False'} : Bool;
      btnInitTagByBodyType1Pls { ExternalAccessible := 'False'; ExternalVisible := 'False'; ExternalWritable := 'False'} : Bool;
      btnInitTagByPopIdEdg { ExternalAccessible := 'False'; ExternalVisible := 'False'; ExternalWritable := 'False'} : Bool;
      btnInitTagByPopIdPls { ExternalAccessible := 'False'; ExternalVisible := 'False'; ExternalWritable := 'False'} : Bool;
      btnRplcTagByMixNbrEdg { ExternalAccessible := 'False'; ExternalVisible := 'False'; ExternalWritable := 'False'} : Bool;
      btnRplcTagByMixNbrPls { ExternalAccessible := 'False'; ExternalVisible := 'False'; ExternalWritable := 'False'} : Bool;
      btnRplcTagByMixNbrEnable { ExternalAccessible := 'False'; ExternalVisible := 'False'; ExternalWritable := 'False'} : Word;
      btnRplcTagByTagIDEdg { ExternalAccessible := 'False'; ExternalVisible := 'False'; ExternalWritable := 'False'} : Bool;
      btnRplcTagByTagIDPls { ExternalAccessible := 'False'; ExternalVisible := 'False'; ExternalWritable := 'False'} : Bool;
      btnRplcTagByTagIDEnable { ExternalAccessible := 'False'; ExternalVisible := 'False'; ExternalWritable := 'False'} : Word;
      btnRplcTagByBodyIdEdg { ExternalAccessible := 'False'; ExternalVisible := 'False'; ExternalWritable := 'False'} : Bool;
      btnRplcTagByBodyIdPls { ExternalAccessible := 'False'; ExternalVisible := 'False'; ExternalWritable := 'False'} : Bool;
      btnRplcTagByBodyIdEnable { ExternalAccessible := 'False'; ExternalVisible := 'False'; ExternalWritable := 'False'} : Word;
      btnRplcTagByPopIDEdg { ExternalAccessible := 'False'; ExternalVisible := 'False'; ExternalWritable := 'False'} : Bool;
      btnRplcTagByPopIDPls { ExternalAccessible := 'False'; ExternalVisible := 'False'; ExternalWritable := 'False'} : Bool;
      btnRplcTagByPopIDEnable { ExternalAccessible := 'False'; ExternalVisible := 'False'; ExternalWritable := 'False'} : Word;
      GetVEMDataByRFIDBeginReq1 { ExternalAccessible := 'False'; ExternalVisible := 'False'; ExternalWritable := 'False'} : Bool;
      GetVEMDataByRFIDBeginReq2 { ExternalAccessible := 'False'; ExternalVisible := 'False'; ExternalWritable := 'False'} : Bool;
      GetVEMDataByRFIDBeginReq3 { ExternalAccessible := 'False'; ExternalVisible := 'False'; ExternalWritable := 'False'} : Bool;
      InteractEnable { ExternalAccessible := 'False'; ExternalVisible := 'False'; ExternalWritable := 'False'} : Bool;   // Interactions enabled
      Status { ExternalAccessible := 'False'; ExternalVisible := 'False'; ExternalWritable := 'False'} : Int;
      TriggOnTimerElapsed { ExternalAccessible := 'False'; ExternalVisible := 'False'; ExternalWritable := 'False'} : Bool;   // Antenna trigger - On
      AntennaTriggOnTimeAct { ExternalAccessible := 'False'; ExternalVisible := 'False'; ExternalWritable := 'False'} : DInt;
      TriggerOffTimerElapsed { ExternalAccessible := 'False'; ExternalVisible := 'False'; ExternalWritable := 'False'} : Bool;   // Antenna trigger - Off
      AntennaTriggOffTimeAct { ExternalAccessible := 'False'; ExternalVisible := 'False'; ExternalWritable := 'False'} : DInt;
      AntennaTrigg { ExternalAccessible := 'False'; ExternalVisible := 'False'; ExternalWritable := 'False'} : Bool;
      AntennaTriggCntr { ExternalAccessible := 'False'; ExternalVisible := 'False'; ExternalWritable := 'False'} : Int;   // Antenna trigger - Counter
      AntennaStatus { ExternalAccessible := 'False'; ExternalVisible := 'False'; ExternalWritable := 'False'} : Int;
      StartReadEdg { ExternalAccessible := 'False'; ExternalVisible := 'False'; ExternalWritable := 'False'} : Bool;
      StartReadPls { ExternalAccessible := 'False'; ExternalVisible := 'False'; ExternalWritable := 'False'} : Bool;
      StartInitTagEdg { ExternalAccessible := 'False'; ExternalVisible := 'False'; ExternalWritable := 'False'} : Bool;
      StartInitTagPls { ExternalAccessible := 'False'; ExternalVisible := 'False'; ExternalWritable := 'False'} : Bool;
      Alarm { ExternalAccessible := 'False'; ExternalVisible := 'False'; ExternalWritable := 'False'} : Bool;
      BodyIdMemReplaceTag { ExternalAccessible := 'False'; ExternalVisible := 'False'; ExternalWritable := 'False'} : DWord;
      MixNbrMemReplaceTag { ExternalAccessible := 'False'; ExternalVisible := 'False'; ExternalWritable := 'False'} : DWord;
      PopIdMemReplaceTag { ExternalAccessible := 'False'; ExternalVisible := 'False'; ExternalWritable := 'False'} : DWord;
      PopIdSuffixMemReplaceTag { ExternalAccessible := 'False'; ExternalVisible := 'False'; ExternalWritable := 'False'} : Char;
      PopTypeMemReplaceTag { ExternalAccessible := 'False'; ExternalVisible := 'False'; ExternalWritable := 'False'} : DWord;
      TagIdMem { ExternalAccessible := 'False'; ExternalVisible := 'False'; ExternalWritable := 'False'} : DWord;
      TagIdMemReplaceTag { ExternalAccessible := 'False'; ExternalVisible := 'False'; ExternalWritable := 'False'} : DWord;
      TagIdMemReplaceTagStr { ExternalAccessible := 'False'; ExternalVisible := 'False'; ExternalWritable := 'False'} : String[7];
      BodyIDMemInit { ExternalAccessible := 'False'; ExternalVisible := 'False'; ExternalWritable := 'False'} : DWord;
      BodyType1MemInit { ExternalAccessible := 'False'; ExternalVisible := 'False'; ExternalWritable := 'False'} : DWord;
      PopIDMemInit { ExternalAccessible := 'False'; ExternalVisible := 'False'; ExternalWritable := 'False'} : DWord;
      PopIDSuffixMemInit { ExternalAccessible := 'False'; ExternalVisible := 'False'; ExternalWritable := 'False'} : Char;
      PopTypeMemInit { ExternalAccessible := 'False'; ExternalVisible := 'False'; ExternalWritable := 'False'} : DWord;
      StartTriggOnTimer { ExternalAccessible := 'False'; ExternalVisible := 'False'; ExternalWritable := 'False'} : Bool;   // Trigger on timer - Start
      StartTriggOffTimer { ExternalAccessible := 'False'; ExternalVisible := 'False'; ExternalWritable := 'False'} : Bool;   // Trigger off timer - Start
      TempDiv { ExternalAccessible := 'False'; ExternalVisible := 'False'; ExternalWritable := 'False'} : DInt;   // Temporary divider
      TempDInt { ExternalAccessible := 'False'; ExternalVisible := 'False'; ExternalWritable := 'False'} : DInt;
      TempReal { ExternalAccessible := 'False'; ExternalVisible := 'False'; ExternalWritable := 'False'} : Real;
      _TriggOnTmr { ExternalAccessible := 'False'; ExternalVisible := 'False'; ExternalWritable := 'False'; S7_SetPoint := 'True'} : "LTimer";   // FB / Trigger on timer
      _TriggOffTmr { ExternalAccessible := 'False'; ExternalVisible := 'False'; ExternalWritable := 'False'; S7_SetPoint := 'True'} : "LTimer";   // FB / Trigger off timer
   END_VAR
   VAR CONSTANT
      TAG_ID_LENGTH_MAX : Int := 7;
      CMD_INIT_TAG : DWord := 2003;   // Command code - Init tag
      CMD_REPLACE_TAG : DWord := 2002;   // Command code - Replace tag
      ANTENNA_TRIGG_CNTR_MAX : Int := 3;   // Maximum amount of triggers
      STATUS_000 : Int;   // Status 000 : No action
      STATUS_001 : Int := 1;   // Status 001 : Success
      STATUS_002 : Int := 2;   // Status 002 : Busy
      STATUS_MINUS_001 : Int := -1;   // Status - 001 : No signal from RFID antenna
      STATUS_MINUS_002 : Int := -2;   // Status - 002 : Tag read error
      STATUS_MINUS_008 : Int := -12;   // Status - 008 : Sequence overtime
      STATUS_MINUS_100 : Int := -100;   // Status - 100 : TagId does not exist
      OFF : Word := 16#0000;   // HMI animation - No animation
      VISIBLE : Word := 16#0001;   // HMI animation - Visible
      ENABLE : Word := 16#0002;   // HMI animation - Enable
      COLOUR_DEFAULT : Word := 16#0000;   // HMI animation - Default colour
      COLOUR_RED : Word := 16#0010;   // HMI animation - Colour red
      COLOUR_GREEN : Word := 16#0020;   // HMI animation - Colour green
      COLOUR_BLUE : Word := 16#0040;   // HMI animation - Colour blue
      COLOUR_WHITE : Word := 16#0080;   // HMI animation - Colour white
      SECTION_HMI : Bool := TRUE;
      SECTION_OUTPUTS : Bool := TRUE;
   END_VAR
BEGIN
   (******************************************************************************
    Changelog

       17W23D1 18:00H PMo
       - Conversion from FBD TO SCL

    List OF authors

       Company : Volvo Cars Gent
       Name    : Patrick Moreau (PMo)
       E-mail  : patrick.moreau@volvocars.com
       Tel.    : +32 9 2503165

    Description

       This module is part OF the VIDS suite and is used to read, initialize and 
       replace the RFID.
       To use this module, VIDSMaster is required

    ******************************************************************************)

   (******************************************************************************)
   (* Alarm                                                                      *)
   (******************************************************************************)
   IF NOT #I_AntennaStatus AND NOT #IO_VIDS.GetVEMDataByRFID.Running AND FALSE THEN        //Check antenna
       #Status := #STATUS_MINUS_001;   //No signal from RFID antenna
   END_IF;
   IF #I_AntennaStatus AND #Status = #STATUS_MINUS_001 AND FALSE THEN
       #Status := #STATUS_000;
   END_IF;

   (******************************************************************************)
   (* Create pulses                                                              *)
   (******************************************************************************)

   //Start read - Create pulse
   #StartReadPls := #I_StartRead AND NOT #StartReadEdg;
   #StartReadEdg := #I_StartRead;

   //< Force read > button - Create pulse
   #btnForceReadPls := #H_RFID.H_btnForceRead <> 0 AND NOT #btnForceReadEdg;
   #btnForceReadEdg := #H_RFID.H_btnForceRead <> 0;

   //Start init - Create pulse
   #StartInitTagPls := #I_StartInitTag AND NOT #StartInitTagEdg;
   #StartInitTagEdg := #I_StartInitTag;

   // < Start Init tag BY BodyID > button - Create pulse
   #btnInitTagByBodyIdPls := (#H_RFID.H_btnInitTagByBodyId <> 0) AND NOT #btnInitTagByBodyIdEdg;
   #btnInitTagByBodyIdEdg := (#H_RFID.H_btnInitTagByBodyId <> 0);

   // < Start Init tag BY BodyType1 > button - Create pulse
   #btnInitTagByBodyType1Pls := (#H_RFID.H_btnInitTagByBodyType1 <> 0) AND NOT #btnInitTagByBodyType1Edg;
   #btnInitTagByBodyType1Edg := (#H_RFID.H_btnInitTagByBodyType1 <> 0);

   // < Start Init tag BY PopID > button - Create pulse
   #btnInitTagByPopIdPls := (#H_RFID.H_btnInitTagByPopId <> 0) AND NOT #btnInitTagByPopIdEdg;
   #btnInitTagByPopIdEdg := (#H_RFID.H_btnInitTagByPopId <> 0);

   //< Replace Tag BY TagID > button - Create pulse
   #btnRplcTagByTagIDPls := #H_RFID.H_btnRplcTagByTagID <> 0 AND NOT #btnRplcTagByTagIDEdg;
   #btnRplcTagByTagIDEdg := #H_RFID.H_btnRplcTagByTagID <> 0;

   //< Replace Tag BY BodyID > button - Create pulse
   #btnRplcTagByBodyIdPls := #H_RFID.H_btnRplcTagByBodyId <> 0 AND NOT #btnRplcTagByBodyIdEdg;
   #btnRplcTagByBodyIdEdg := #H_RFID.H_btnRplcTagByBodyId <> 0;

   //< Replace Tag BY Mixnumber > button - Create pulse
   #btnRplcTagByMixNbrPls := #H_RFID.H_btnRplcTagByMIxNbr <> 0 AND NOT #btnRplcTagByMixNbrEdg;
   #btnRplcTagByMixNbrEdg := #H_RFID.H_btnRplcTagByMIxNbr <> 0;

   //< Replace Tag BY PopId > button - Create pulse
   #btnRplcTagByPopIDPls := #H_RFID.H_btnRplcTagByPopId <> 0 AND NOT #btnRplcTagByPopIDEdg;
   #btnRplcTagByPopIDEdg := #H_RFID.H_btnRplcTagByPopId <> 0;

   (******************************************************************************)
   (* Get VEM data by RFID - Begin request                                       *)
   (******************************************************************************)

   //By Read
   #GetVEMDataByRFIDBeginReq1 := #I_AntennaStatus AND (#StartReadPls OR #btnForceReadPls);

   //By Replace tag
   IF  #btnRplcTagByTagIDPls THEN
       #TagIdMemReplaceTag := #H_RFID.H_txtTagIDRplcTag;
       #BodyIdMemReplaceTag := 0;
       #MixNbrMemReplaceTag := 0;
       #PopIdMemReplaceTag := 0;
       #PopIdSuffixMemReplaceTag := ' ';
       #PopTypeMemReplaceTag := 0;
       #StartReplaceTagMem := TRUE;
   ELSIF  #btnRplcTagByBodyIdPls THEN
       #TagIdMemReplaceTag := 0;
       #BodyIdMemReplaceTag := #H_RFID.H_txtBodyIDRplcTag;
       #MixNbrMemReplaceTag := 0;
       #PopIdMemReplaceTag := 0;
       #PopIdSuffixMemReplaceTag := ' ';
       #PopTypeMemReplaceTag := 0;
       #StartReplaceTagMem := TRUE;
   ELSIF  #btnRplcTagByMixNbrPls THEN
       #TagIdMemReplaceTag :=0;
       #BodyIdMemReplaceTag := 0;
       #MixNbrMemReplaceTag := #H_RFID.H_txtMixNbrRplcTag;
       #PopIdMemReplaceTag := 0;
       #PopIdSuffixMemReplaceTag := ' ';
       #PopTypeMemReplaceTag := 0;
       #StartReplaceTagMem := TRUE;
   ELSIF  #btnRplcTagByPopIDPls THEN
       #TagIdMemReplaceTag := 0;
       #BodyIdMemReplaceTag := 0;
       #MixNbrMemReplaceTag := 0;
       #PopIdMemReplaceTag := #H_RFID.H_txtPopIDRplcTag;
       #PopIdSuffixMemReplaceTag := #H_RFID.H_txtPopIDSuffixRplcTag;
       #PopTypeMemReplaceTag := #H_RFID.H_txtPopTypeRplcTag;
       #StartReplaceTagMem := TRUE;
   END_IF;
   #GetVEMDataByRFIDBeginReq2 := #btnRplcTagByTagIDPls OR #btnRplcTagByBodyIdPls OR #btnRplcTagByMixNbrPls OR #btnRplcTagByPopIDPls;

   //By Init tag
   IF  #StartInitTagPls THEN
       IF #I_BodyIDInitTag <> 0 THEN
           #BodyIDMemInit := #I_BodyIDInitTag;
           #BodyType1MemInit := 0;
           #PopIDMemInit := 0;
           #PopIDSuffixMemInit := ' ';
           #PopTypeMemInit := 0;
       ELSIF #I_BodyType1InitTag <> 0 THEN
           #BodyIDMemInit := 0;
           #PopIDMemInit := 0;
           #PopIDSuffixMemInit := ' ';
           #PopTypeMemInit := 0;
           #BodyType1MemInit := #I_BodyType1InitTag;
       ELSIF #I_PopIDInitTag <> 0 THEN
           #BodyIDMemInit := 0;
           #BodyType1MemInit := 0;
           #PopIDMemInit := #I_PopIDInitTag;
           #PopIDSuffixMemInit := #I_PopIDSuffixInitTag;
           #PopTypeMemInit := #I_PopTypeInitTag;
       END_IF;
       #StartInitMem := TRUE;
   ELSIF  #btnInitTagByBodyIdPls THEN
       #BodyIDMemInit := #H_RFID.H_txtBodyIDInitTag;
       #BodyType1MemInit := 0;
       #PopIDMemInit := 0;
       #PopIDSuffixMemInit := ' ';
       #PopTypeMemInit := 0;
       #StartInitMem := TRUE;
   ELSIF #I_AntennaStatus AND #btnInitTagByBodyType1Pls THEN
       #BodyIDMemInit := 0;
       #PopIDMemInit := 0;
       #PopIDSuffixMemInit := ' ';
       #PopTypeMemInit := 0;
       #BodyType1MemInit := #H_RFID.H_txtBodyType1InitTag;
       #StartInitMem := TRUE;
   ELSIF #I_AntennaStatus AND #btnInitTagByPopIdPls THEN
       #BodyIDMemInit := 0;
       #BodyType1MemInit := 0;
       #PopIDMemInit := #H_RFID.H_txtPopIdInitTag;
       #PopIDSuffixMemInit := #H_RFID.H_txtPopIdSuffixInitTag;
       #PopTypeMemInit := #H_RFID.H_txtPopTypeInitTag;
       #StartInitMem := TRUE;
   END_IF;

   #GetVEMDataByRFIDBeginReq3 := #StartInitTagPls OR #btnInitTagByBodyIdPls OR #btnInitTagByBodyType1Pls OR #btnInitTagByPopIdPls;

   //Begin request - Summary
   #IO_VIDS.GetVEMDataByRFID.BeginReq := #IO_VIDS.PartPres  AND
   (#GetVEMDataByRFIDBeginReq1 OR #GetVEMDataByRFIDBeginReq2 OR #GetVEMDataByRFIDBeginReq3) AND NOT 
   #IO_VIDS.GetVEMDataByRFID.Running;

   //Reset when not part present
   IF NOT #IO_VIDS.PartPres THEN

       #StartReplaceTagMem := FALSE;
       #StartInitMem := FALSE;

   END_IF;

   #Reset := NOT #IO_VIDS.PartPres OR #IO_VIDS.GetVEMDataByRFID.BeginReq OR #IO_VIDS.InitTag.BeginReq OR #IO_VIDS.ReplaceTag.BeginReq;

   IF  #Reset THEN



       #ReadOK := FALSE;
       #ReadNOK := FALSE;
       #InitTagOK := FALSE;
       #InitTagNOK := FALSE;
       #ReplaceTagOK := FALSE;
       #ReplaceTagNOK := FALSE;
       #AntennaStatus := 0;
       #Status := 0;

   END_IF;

   (******************************************************************************)
   (* Get VEM data by RFID - Begin                                               *)
   (******************************************************************************)

   //Activate antenna
   IF #IO_VIDS.GetVEMDataByRFID.OkBegin THEN
       #Status := #STATUS_002;             //Set Status busy

       #AntennaTriggCntr := 0;             //Reset antenna trigger Counter
       #StartTriggOnTimer := TRUE;         //Start trigger
   END_IF;

   //Step 0 On Active - Get VEM Data - Begin
   #IO_VIDS.GetVEMDataByRFID.Begin := #IO_VIDS.GetVEMDataByRFID.OkBegin;

   (******************************************************************************)
   (* Get VEM data by RFID - Antenna triggering                                  *)
   (******************************************************************************)

   IF NOT #I_AntennaStatus THEN
       #StartTriggOnTimer := FALSE;
       #StartTriggOffTimer := FALSE;
   END_IF;

   //Antenna Trigger on timer
   #_TriggOnTmr(I_StartTimer := #StartTriggOnTimer,
                I_HoldTimer := FALSE,
                I_MaxTimerValue := #C_AntennaTriggOnTime,
                O_TimerResult => #TriggOnTimerElapsed,
                O_TimerValue => #AntennaTriggOnTimeAct);

   //Start off timer
   IF #TriggOnTimerElapsed THEN
       #StartTriggOnTimer := FALSE;
       #StartTriggOffTimer := TRUE;
   END_IF;

   //Antenna Trigger off timer
   #_TriggOffTmr(I_StartTimer := #StartTriggOffTimer,
                 I_HoldTimer := FALSE,
                 I_MaxTimerValue := #C_AntennaTriggOffTime,
                 O_TimerResult => #TriggerOffTimerElapsed,
                 O_TimerValue => #AntennaTriggOffTimeAct);

   //Restart trigger timer
   IF #TriggerOffTimerElapsed THEN
       #AntennaTriggCntr := #AntennaTriggCntr + 1;
       IF #AntennaTriggCntr < #ANTENNA_TRIGG_CNTR_MAX THEN
           #StartTriggOffTimer := FALSE;
           #StartTriggOnTimer := TRUE;
       ELSE
           #StartTriggOnTimer := FALSE;
           #StartTriggOffTimer := FALSE;
           #AntennaStatus := #STATUS_MINUS_002;
       END_IF;
   END_IF;

   //Antenna Trigger
   #AntennaTrigg := #StartTriggOnTimer AND NOT #TriggOnTimerElapsed AND #I_AntennaStatus;

   (******************************************************************************)
   (* Get VEM data by RFID - Finish                                              *)
   (******************************************************************************)

   //Make sure we create a pulse
   #IO_VIDS.ReplaceTag.BeginReq := FALSE;
   #IO_VIDS.InitTag.BeginReq := FALSE;

   //Get VEMData by RFID - Finished
   IF #IO_VIDS.GetVEMDataByRFID.Finished THEN

       //Antenna status has priority
       IF #AntennaStatus < 0 THEN
           #Status := #AntennaStatus;
       ELSE
           #Status := #IO_VIDS.GetVEMDataByRFID.Status;
       END_IF;

       //Read OK or NOK
       IF #Status = 1 THEN
           #ReadOK := True;
       ELSE
           #ReadNOK := True;
       END_IF;

       //Replace tag
       IF #StartReplaceTagMem THEN
           #StartReplaceTagMem := FALSE;
           IF #Status <> #STATUS_MINUS_002 THEN
               #TagIdMem := #IO_VIDS.VEMData.Identification;
               #IO_VIDS.ReplaceTag.BeginReq := TRUE;       //Replace tag - Begin request
           END_IF;

       //Init tag
       ELSIF #StartInitMem THEN
           #StartInitMem := FALSE;
           IF #Status <> #STATUS_MINUS_002 THEN
               #TagIdMem := #IO_VIDS.VEMData.Identification;
               #IO_VIDS.InitTag.BeginReq := TRUE;
           END_IF;
       END_IF;

   END_IF;

   (******************************************************************************)
   (* Replace tag - Begin & Finished                                             *)
   (******************************************************************************)

   IF #IO_VIDS.ReplaceTag.OkBegin THEN

       #Status := #STATUS_002;             //Set Status busy
       #IO_VIDS.VEMData.CommandCode := #CMD_REPLACE_TAG;
       #IO_VIDS.VEMData.Identification := #TagIdMem;

       IF #TagIdMemReplaceTag <> 0 THEN
           //TagId in specificdata
           #TempDInt := DWORD_TO_DINT(#TagIdMemReplaceTag);
           #TempReal := DINT_TO_REAL(#TAG_ID_LENGTH_MAX-1);
           #TempDiv := REAL_TO_DINT(10 ** #TempReal);
           FOR #i := 0 TO (#TAG_ID_LENGTH_MAX-1) DO
               #IO_VIDS.SpecificDataInit[#i] := DINT_TO_CHAR(#TempDInt / #TempDiv + 48);
               #TempDInt := #TempDInt MOD #TempDiv;
               #TempDiv := #TempDiv / 10;
           END_FOR;
           #IO_VIDS.VEMData.SpecificDataLength := DINT_TO_DWORD(#TAG_ID_LENGTH_MAX);
       ELSE
           #IO_VIDS.VEMData.BodyID := #BodyIdMemReplaceTag;
           #IO_VIDS.VEMData.MixNumber := #MixNbrMemReplaceTag;
           #IO_VIDS.VEMData.PopID := #PopIdMemReplaceTag;
           #IO_VIDS.VEMData.PopIDSuffix := #PopIdSuffixMemReplaceTag;
           #IO_VIDS.VEMData.PopType := #PopTypeMemReplaceTag;
           #IO_VIDS.VEMData.SpecificDataLength := 0;
       END_IF;

   ELSIF #IO_VIDS.ReplaceTag.Finished THEN
       #Status := #IO_VIDS.ReplaceTag.Status;
       IF #Status = 1 THEN
           #ReplaceTagOK := True;
       ELSE
           #ReplaceTagNOK := True;
       END_IF;
   END_IF;

   #IO_VIDS.ReplaceTag.Begin := #IO_VIDS.ReplaceTag.OkBegin;

   (******************************************************************************)
   (* Init tag - Begin & Finished                                                *)
   (******************************************************************************)

   IF #IO_VIDS.InitTag.OkBegin THEN

       #Status := #STATUS_002;             //Set Status busy
       #IO_VIDS.VEMData.Identification := #TagIdMem;
       #IO_VIDS.VEMData.BodyID := #BodyIDMemInit;
       #IO_VIDS.VEMData.BodyType1 := #BodyType1MemInit;
       #IO_VIDS.VEMData.PopID := #PopIDMemInit;
       #IO_VIDS.VEMData.PopIDSuffix := #PopIDSuffixMemInit;
       #IO_VIDS.VEMData.PopType := #PopTypeMemInit;

       #IO_VIDS.VEMData.CommandCode := #CMD_INIT_TAG;

   ELSIF #IO_VIDS.InitTag.Finished THEN
       #Status := #IO_VIDS.InitTag.Status;
       IF #Status = 1 THEN
           #InitTagOK := True;
       ELSE
           #InitTagNOK := True;
       END_IF;
   END_IF;

   #IO_VIDS.InitTag.Begin := #IO_VIDS.InitTag.OkBegin;

   (******************************************************************************)
   (* Alarm = status <0                                                          *)
   (******************************************************************************)
   IF #Status < 0 THEN
       #Alarm := TRUE;
   ELSE
       #Alarm := false;
   END_IF;

   "LAlarmSummary"(I_AlarmA := "FALSE",
                   I_AlarmB := "FALSE",
                   I_AlarmC := #Alarm,
                   I_AlarmD := "FALSE",
                   I_AlarmABCondition := "FALSE",
                   IO_Alarm := #IO_Alarm,
                   C_UpperLevelHW := "FALSE",
                   C_UpperLevelSafety := "FALSE",
                   C_Safety := "FALSE",
                   C_Mechanic := "FALSE",
                   C_Transport := "FALSE",
                   C_Feature1 := "FALSE",
                   C_Feature2 := "FALSE",
                   C_Feature3 := "FALSE");

   (******************************************************************************)
   (* Outputs                                                                    *)
   (******************************************************************************)
   IF #SECTION_OUTPUTS THEN

       #O_AntennaTrigg := #AntennaTrigg;                   //Antenna Trigger

       #O_Busy := #IO_VIDS.GetVEMDataByRFID.Running;       //Read Busy
       #O_ReadOK := #ReadOK;                               //Read OK
       #O_ReadNOK := #ReadNOK;                             //Read NOK

       #O_InitTagBusy := #IO_VIDS.InitTag.Running;         //Init tag busy
       #O_InitTagOK := #InitTagOK;                         //Init OK
       #O_InitTagNOK := #InitTagNOK;                       //Init NOK

       #O_ReplaceTagBusy := #IO_VIDS.ReplaceTag.Running;   //Replace tag busy
       #O_ReplaceTagOK := #ReplaceTagOK;                   //Replace OK
       #O_ReplaceTagNOK := #ReplaceTagNOK;                 //Replace NOK

       #O_Status := #Status;                               //Status
       #O_Alarm := #Status < 0;                            //Alarm

   END_IF;
   (******************************************************************************)
   (* HMI                                                                        *)
   (******************************************************************************)

   IF #SECTION_HMI THEN

       #InteractEnable := #IO_VIDS.PartPres AND NOT #IO_VIDS.GetVEMDataByRFID.Running AND NOT #IO_VIDS.ReplaceTag.Running AND NOT #IO_VIDS.InitTag.Running;

       //HMI - IDType
       IF #IO_VIDS.IDType = 0 THEN
           #H_RFID.H_msgVEMDataBody := #VISIBLE;
           #H_RFID.H_msgVEMDataCarrier := #OFF;
       ELSE
           #H_RFID.H_msgVEMDataBody := #OFF;
           #H_RFID.H_msgVEMDataCarrier := #VISIBLE;
       END_IF;

       //HMI - Message - Part Present - Visible
       IF #IO_VIDS.PartPres THEN
           #H_RFID.H_msgPartPresAnim := #VISIBLE;
       ELSE
           #H_RFID.H_msgPartPresAnim := #OFF;
       END_IF;

       //HMI - VEM Data Valid
       IF #IO_VIDS.VEMDataValid THEN
           #H_RFID.H_msgVEMDataValidAnim := #VISIBLE;
       ELSE
           #H_RFID.H_msgVEMDataValidAnim := #OFF;
       END_IF;

       //HMI - VEM Data NOT Valid
       IF #IO_VIDS.VEMDataNotValid THEN
           #H_RFID.H_msgVEMDataNotValidAnim := #VISIBLE;
       ELSE
           #H_RFID.H_msgVEMDataNotValidAnim := #OFF;
       END_IF;

       //HMI - Status
       #H_RFID.H_msgStatus := #Status;

       //HMI - Antenna ready
       IF #I_AntennaStatus THEN
           #H_RFID.H_indReadyAnim := #VISIBLE;
       ELSE
           #H_RFID.H_indReadyAnim := #OFF;
       END_IF;

       //HMI - Read OK
       IF #ReadOK THEN
           #H_RFID.H_msgReadOkAnim := #VISIBLE;
       ELSE
           #H_RFID.H_msgReadOkAnim := 0;
       END_IF;

       //HMI - Read NOK
       IF #ReadNOK THEN
           #H_RFID.H_msgReadNokAnim := #VISIBLE;
       ELSE
           #H_RFID.H_msgReadNokAnim := 0;
       END_IF;

       //HMI - Replace tag OK
       IF #ReplaceTagOK THEN
           #H_RFID.H_msgRplcTagOkAnim := #VISIBLE;
       ELSE
           #H_RFID.H_msgRplcTagOkAnim := 0;
       END_IF;

       //HMI - Replace tag NOK
       IF #ReplaceTagNOK THEN
           #H_RFID.H_msgRplcTagNokAnim := #VISIBLE;
       ELSE
           #H_RFID.H_msgRplcTagNokAnim := 0;
       END_IF;

       //HMI - Init tag OK
       IF #InitTagOK THEN
           #H_RFID.H_msgInitTagOkAnim := #VISIBLE;
       ELSE
           #H_RFID.H_msgInitTagOkAnim := 0;
       END_IF;

       //HMI - Init tag NOK
       IF #InitTagNOK THEN
           #H_RFID.H_msgInitTagNokAnim := #VISIBLE;
       ELSE
           #H_RFID.H_msgInitTagNokAnim := 0;
       END_IF;

       //HMI - Animation Antenna Status
       IF #I_AntennaStatus THEN
           #H_RFID.H_indAntennaStatusAnim := 1;
       ELSE
           #H_RFID.H_indAntennaStatusAnim := 0;
       END_IF;

       //HMI - Animation Antenna Trigger
       IF #AntennaTrigg THEN
           #H_RFID.H_indAntennaTriggAnim := #VISIBLE;
       ELSE
           #H_RFID.H_indAntennaTriggAnim := #OFF;
       END_IF;


   (******************************************************************************)
   (* HMI - Text fields                                                          *)
   (******************************************************************************)

       //HMI - ReplaceTag - Reset Values
       IF NOT #IO_VIDS.PartPres OR (#IO_VIDS.GetVEMDataByRFID.BeginReq AND NOT #StartReplaceTagMem) THEN
           #H_RFID.H_txtTagIDRplcTag := 0;
           #H_RFID.H_txtBodyIDRplcTag := 0;
           #H_RFID.H_txtMixNbrRplcTag := 0;
           #H_RFID.H_txtPopIDRplcTag := 0;
           #H_RFID.H_txtPopIDSuffixRplcTag := ' ';
           #H_RFID.H_txtPopTypeRplcTag := 0;
       END_IF;

       IF #InteractEnable THEN
           #H_RFID.H_txtTagIDRplcTagAnim := #VISIBLE OR #ENABLE OR #COLOUR_WHITE;  //HMI - txtTagIDReplaceTag - Animation
           #H_RFID.H_txtBodyIDRplcTagAnim := #VISIBLE OR #ENABLE OR #COLOUR_WHITE;  //HMI - txtBodyIDReplaceTag - Animation
           #H_RFID.H_txtMixNbrRplcTagAnim := #VISIBLE OR #ENABLE OR #COLOUR_WHITE; //HMI - txtMixNbrReplaceTag - Animation
           #H_RFID.H_txtPopIDRplcTagAnim := #VISIBLE OR #ENABLE OR #COLOUR_WHITE; //HMI - txtPopIdReplaceTag - Animation
           #H_RFID.H_txtPopIDSuffixRplcTagAnim := #VISIBLE OR #ENABLE OR #COLOUR_WHITE; //HMI - txtPopIdSuffixReplaceTag - Animation
           #H_RFID.H_txtPopTypeRplcTagAnim := #VISIBLE OR #ENABLE OR #COLOUR_WHITE; //HMI - txtPopTypeReplaceTag - Animation
       ELSE
           #H_RFID.H_txtTagIDRplcTagAnim := #VISIBLE OR #COLOUR_DEFAULT;  //HMI - txtTagIDReplaceTag - Animation
           #H_RFID.H_txtBodyIDRplcTagAnim := #VISIBLE OR #COLOUR_DEFAULT;  //HMI - txtBodyIDReplaceTag - Animation
           #H_RFID.H_txtMixNbrRplcTagAnim := #VISIBLE OR #COLOUR_DEFAULT; //HMI - txtMixNbrReplaceTag - Animation
           #H_RFID.H_txtPopIDRplcTagAnim := #VISIBLE OR #COLOUR_DEFAULT; //HMI - txtPopIdReplaceTag - Animation
           #H_RFID.H_txtPopIDSuffixRplcTagAnim := #VISIBLE OR #COLOUR_DEFAULT; //HMI - txtPopIdSuffixReplaceTag - Animation
           #H_RFID.H_txtPopTypeRplcTagAnim := #VISIBLE OR #COLOUR_DEFAULT; //HMI - txtPopTypeReplaceTag - Animation
       END_IF;


       //HMI - InitTag - Reset Values
       IF NOT #IO_VIDS.PartPres OR (#IO_VIDS.GetVEMDataByRFID.BeginReq AND NOT #StartInitMem) THEN
           #H_RFID.H_txtBodyIDInitTag := 0;
           #H_RFID.H_txtBodyType1InitTag := 0;
           #H_RFID.H_txtPopIdInitTag := 0;
           #H_RFID.H_txtPopIdSuffixInitTag := ' ';
           #H_RFID.H_txtPopTypeInitTag := 0;
       END_IF;

       //HMI - InitTag
       IF #I_InitTagEn  THEN
           IF #InteractEnable THEN
               #H_RFID.H_txtBodyIDInitTagAnim := #VISIBLE OR #ENABLE OR #COLOUR_WHITE;     //HMI - txtBodyIDInitTag - Animation
               #H_RFID.H_txtBodyType1InitTagAnim := #VISIBLE OR #ENABLE OR #COLOUR_WHITE;  //HMI - txtBodyType1InitTag - Animation
               #H_RFID.H_txtPopIdInitTagAnim := #VISIBLE OR #ENABLE OR #COLOUR_WHITE;      //HMI - txtPopIdInitTag - Animation
               #H_RFID.H_txtPopIdSuffixInitTagAnim := #VISIBLE OR #ENABLE OR #COLOUR_WHITE;//HMI - txtPopIdSuffixInitTag - Animation
               #H_RFID.H_txtPopTypeInitTagAnim := #VISIBLE OR #ENABLE OR #COLOUR_WHITE;    //HMI - txtPopTypeInitTag - Animation
           ELSE
               #H_RFID.H_txtBodyIDInitTagAnim := #VISIBLE OR #COLOUR_DEFAULT;     //HMI - txtBodyIDInitTag - Animation
               #H_RFID.H_txtBodyType1InitTagAnim := #VISIBLE OR #COLOUR_DEFAULT;  //HMI - txtBodyType1InitTag - Animation
               #H_RFID.H_txtPopIdInitTagAnim := #VISIBLE OR #COLOUR_DEFAULT;      //HMI - txtPopIdInitTag - Animation
               #H_RFID.H_txtPopIdSuffixInitTagAnim := #VISIBLE OR #COLOUR_DEFAULT;//HMI - txtPopIdSuffixInitTag - Animation
               #H_RFID.H_txtPopTypeInitTagAnim := #VISIBLE OR #COLOUR_DEFAULT;    //HMI - txtPopTypeInitTag - Animation
           END_IF;
       ELSE
           #H_RFID.H_txtBodyIDInitTagAnim := #VISIBLE;         //HMI - txtBodyIDInitTag - Animation
           #H_RFID.H_txtBodyType1InitTagAnim := #VISIBLE;      //HMI - txtBodyType1InitTag - Animation
           #H_RFID.H_txtPopIdInitTagAnim := #VISIBLE;          //HMI - txtPopIdInitTag - Animation
           #H_RFID.H_txtPopIdSuffixInitTagAnim := #VISIBLE;    //HMI - txtPopIdSuffixInitTag - Animation
           #H_RFID.H_txtPopTypeInitTagAnim := #VISIBLE;        //HMI - txtPopTypeInitTag - Animation
       END_IF;

       //VEM data

       #H_RFID.H_txtTagID := #IO_VEMData.Identification;
       #H_RFID.H_txtBodyID := #IO_VEMData.BodyID;                          //HMI - txtBodyNbr - Value
       #H_RFID.H_txtMixNbr := #IO_VEMData.MixNumber;                       //HMI - txtMixnNbr - Value
       #H_RFID.H_txtCarrierID := #IO_VEMData.CarrierID;                    //HMI - txtCarrierID - Value
       #H_RFID.H_txtBodyTypeMatrix := #IO_VEMData.BodyTypeMatrix;          //HMI - txtBodyTypeMatrix - Value
       #H_RFID.H_txtBodyType1 := #IO_VEMData.BodyType1;                    //HMI - txtBodyType1 - Value
       #H_RFID.H_txtPopId := #IO_VEMData.PopID;                            //HMI - txtPopID - Value
       #H_RFID.H_txtPopIdSuffix := #IO_VEMData.PopIDSuffix;                //HMI - txtPopID - Value
       #H_RFID.H_txtPopType := #IO_VEMData.PopType;                        //HMI - txtPopType - Value

       #H_RFID.H_txtCommandCodeSent := #IO_VIDS.CmdCodeSent;               //HMI - CmdCode Sent
       #H_RFID.H_txtCommandCodeRcvd := #IO_VIDS.CmdCodeRcvd;               //HMI - CmdCode Received

   (******************************************************************************)
   (* HMI - Buttons                                                              *)
   (******************************************************************************)

       #H_RFID.H_btnForceReadAnim := #VISIBLE OR #ENABLE;

       //Replace tag
       IF #H_RFID.H_txtTagIDRplcTag <> 0 THEN
           #btnRplcTagByTagIDEnable := #ENABLE;
       ELSE
           #btnRplcTagByTagIDEnable := #OFF;
       END_IF;
       #H_RFID.H_btnRplcTagByTagIDAnim := #VISIBLE OR #btnRplcTagByTagIDEnable;

       //Replace tag
       IF #H_RFID.H_txtBodyIDRplcTag <> 0 THEN
           #btnRplcTagByBodyIdEnable := #ENABLE;
       ELSE
           #btnRplcTagByBodyIdEnable := #OFF;
       END_IF;
       #H_RFID.H_btnRplcTagByBodyIdAnim := #VISIBLE OR #btnRplcTagByBodyIdEnable;

       //Replace tag
       IF #H_RFID.H_txtMixNbrRplcTag <> 0 THEN
           #btnRplcTagByMixNbrEnable := #ENABLE;
       ELSE
           #btnRplcTagByMixNbrEnable := #OFF;
       END_IF;
       #H_RFID.H_btnRplcTagByMixNbrAnim := #VISIBLE OR #btnRplcTagByMixNbrEnable;

       //Replace tag
       IF #H_RFID.H_txtPopIDRplcTag <> 0 THEN
           #btnRplcTagByPopIDEnable := #ENABLE;
       ELSE
           #btnRplcTagByPopIDEnable := #OFF;
       END_IF;
       #H_RFID.H_btnRplcTagByPopIdAnim := #VISIBLE OR #btnRplcTagByPopIDEnable;

       //Init tag
       IF #I_InitTagEn THEN
           #H_RFID.H_btnInitTagByBodyIdAnim := #VISIBLE OR #ENABLE;
           #H_RFID.H_btnInitTagByBodyType1Anim := #VISIBLE OR #ENABLE;
           #H_RFID.H_btnInitTagByPopIdAnim := #VISIBLE OR #ENABLE;
       ELSE
           #H_RFID.H_btnInitTagByBodyIdAnim := #VISIBLE;
           #H_RFID.H_btnInitTagByBodyType1Anim := #VISIBLE;
           #H_RFID.H_btnInitTagByPopIdAnim := #VISIBLE;
       END_IF;

       //HMI Reset buttons
       #H_RFID.H_btnForceRead := 0;
       #H_RFID.H_btnRplcTagByTagID := 0;
       #H_RFID.H_btnRplcTagByBodyId := 0;
       #H_RFID.H_btnRplcTagByMIxNbr := 0;
       #H_RFID.H_btnRplcTagByPopId := 0;
       #H_RFID.H_btnInitTagByBodyId := 0;
       #H_RFID.H_btnInitTagByBodyType1 := 0;
       #H_RFID.H_btnInitTagByPopId := 0;

   (******************************************************************************)
   (* Icon animation                                                             *)
   (******************************************************************************)

       "LIAnimDWord"(I_SetPos := FALSE,
                     I_ResetPos := FALSE,
                     I_Active := #Status > 1,
                     I_Visible := FALSE,
                     I_OutOfUse := FALSE,
                     I_IntlkSet := FALSE,
                     I_IntlkReset := FALSE,
                     I_IntlkSetAlm := FALSE,
                     I_IntlkResetAlm := FALSE,
                     I_ManualMode := FALSE,
                     I_FncSelInHMI := FALSE,
                     I_AnySelected := FALSE,
                     I_AlarmA := FALSE,
                     I_AlarmB := FALSE,
                     I_AlarmC := #Status < 0,
                     I_AlarmD := FALSE,
                     I_SafetyOk := FALSE,
                     I_Service:="TRUE",
                     I_Spare1:="FALSE",
                     I_Spare2:="FALSE",
                     I_Spare3:="FALSE",
                     I_Spare4:="FALSE",
                     I_Spare5:="FALSE",
                     I_Spare6:="FALSE",
                     I_Spare7:="FALSE",
                     I_Spare8:="FALSE",
                     I_Spare9:="FALSE",
                     I_Spare10:="FALSE",
                     I_Spare11:="FALSE",
                     I_Spare12:="FALSE",
                     I_Spare13:="FALSE",
                     I_Spare14:="FALSE",
                     H_IAnim => #H_HMI.H_IAnim);

   END_IF;
END_FUNCTION_BLOCK

FUNCTION_BLOCK "LVIDSTrack"   // FB1205, FBD
TITLE = LVIDS Tracking
{ S7_Optimized_Access := 'TRUE' }
VERSION : 0.1
// stored: AutoNumber false, IsIECCheckEnabled false, IsRetainMemResEnabled false, MemoryReserve 100, SetENOAutomatically False, UDAEnableTagReadback false
   VAR_INPUT
      I_DataModeManEn { ExternalAccessible := 'False'; ExternalVisible := 'False'; ExternalWritable := 'False'} : Bool;   // Data mode manual enabled
      I_OutOfUse { ExternalAccessible := 'False'; ExternalVisible := 'False'; ExternalWritable := 'False'} : Bool;   // Out of use
      I_TagID { ExternalAccessible := 'False'; ExternalVisible := 'False'; ExternalWritable := 'False'} : DInt;   // Tag identification for tracking
      I_BodyID { ExternalAccessible := 'False'; ExternalVisible := 'False'; ExternalWritable := 'False'} : DInt;   // Body identification for tracking
      I_CarrierID { ExternalAccessible := 'False'; ExternalVisible := 'False'; ExternalWritable := 'False'} : DInt;   // Carrier identification for tracking
      I_MixNbr { ExternalAccessible := 'False'; ExternalVisible := 'False'; ExternalWritable := 'False'} : DInt;   // Mixnumber for tracking
      I_BodyType1 { ExternalAccessible := 'False'; ExternalVisible := 'False'; ExternalWritable := 'False'} : DInt;   // Bodytype1 for tracking
      I_PopID { ExternalAccessible := 'False'; ExternalVisible := 'False'; ExternalWritable := 'False'} : UDInt;   // Spare Data / PopID
      I_PopIDSuffix { ExternalAccessible := 'False'; ExternalVisible := 'False'; ExternalWritable := 'False'} : Char;   // PopID suffix
      I_PopType { ExternalAccessible := 'False'; ExternalVisible := 'False'; ExternalWritable := 'False'} : UDInt;   // Pop identifier
      I_Start { ExternalAccessible := 'False'; ExternalVisible := 'False'; ExternalWritable := 'False'} : Bool;   // Start function / Start track
   END_VAR
   VAR_OUTPUT
      O_Ok { ExternalAccessible := 'False'; ExternalVisible := 'False'; ExternalWritable := 'False'} : Bool;   // Function finished / OK
      O_Nok { ExternalAccessible := 'False'; ExternalVisible := 'False'; ExternalWritable := 'False'} : Bool;   // NOK
      O_Busy { ExternalAccessible := 'False'; ExternalVisible := 'False'; ExternalWritable := 'False'} : Bool;   // Busy
      O_Status { ExternalAccessible := 'False'; ExternalVisible := 'False'; ExternalWritable := 'False'} : Int;   // Status ( < 0 : Fault ; 0 : No status; 1 : Success ; > 1 : Busy)
      O_Alarm { ExternalAccessible := 'False'; ExternalVisible := 'False'; ExternalWritable := 'False'} : Bool;   // Alarm
   END_VAR
   VAR_IN_OUT
      IO_VIDS : "VIDS";   // VIDS - internal record
      IO_Alarm : "Alarm";   // Alarm
      H_Track : "H_LVIDSTrack";   // Animation
      H_HMI : "H_HMI";   // Animation
   END_VAR
   VAR
      BtnManTrack { ExternalAccessible := 'False'; ExternalVisible := 'False'; ExternalWritable := 'False'} : Bool;
      BtnManForce { ExternalAccessible := 'False'; ExternalVisible := 'False'; ExternalWritable := 'False'} : Bool;
      BtnManOK { ExternalAccessible := 'False'; ExternalVisible := 'False'; ExternalWritable := 'False'} : Bool;
      BlockAutoStart { ExternalAccessible := 'False'; ExternalVisible := 'False'; ExternalWritable := 'False'} : Bool;
      RSAutoBlock { ExternalAccessible := 'False'; ExternalVisible := 'False'; ExternalWritable := 'False'} : Bool;
      TagIDMem { ExternalAccessible := 'False'; ExternalVisible := 'False'; ExternalWritable := 'False'} : DWord;
      BodyNbrMem { ExternalAccessible := 'False'; ExternalVisible := 'False'; ExternalWritable := 'False'} : DWord;
      MixNbrMem { ExternalAccessible := 'False'; ExternalVisible := 'False'; ExternalWritable := 'False'} : DWord;
      CarrierIDMem { ExternalAccessible := 'False'; ExternalVisible := 'False'; ExternalWritable := 'False'} : DWord;
      BodyType1Mem { ExternalAccessible := 'False'; ExternalVisible := 'False'; ExternalWritable := 'False'} : DWord;
      PopIDMem { ExternalAccessible := 'False'; ExternalVisible := 'False'; ExternalWritable := 'False'} : DWord;
      PopIDSuffixMem { ExternalAccessible := 'False'; ExternalVisible := 'False'; ExternalWritable := 'False'} : Char;
      PopTypeMem { ExternalAccessible := 'False'; ExternalVisible := 'False'; ExternalWritable := 'False'} : DWord;
      StartEdg { ExternalAccessible := 'False'; ExternalVisible := 'False'; ExternalWritable := 'False'} : Bool;   // Edge of start tracking
      StartPls { ExternalAccessible := 'False'; ExternalVisible := 'False'; ExternalWritable := 'False'} : Bool;
      StartTrackEdge2 { ExternalAccessible := 'False'; ExternalVisible := 'False'; ExternalWritable := 'False'} : Bool;   // Edge of start tracking
      StartCmdMem { ExternalAccessible := 'False'; ExternalVisible := 'False'; ExternalWritable := 'False'} : Bool;   // Memory of start command
      FinishPls { ExternalAccessible := 'False'; ExternalVisible := 'False'; ExternalWritable := 'False'} : Bool;   // Pulse of finish tracking
      FinishEdge { ExternalAccessible := 'False'; ExternalVisible := 'False'; ExternalWritable := 'False'} : Bool;   // Edge of finish tracking
      Status { ExternalAccessible := 'False'; ExternalVisible := 'False'; ExternalWritable := 'False'} : Int;   // Status
      Alarm { ExternalAccessible := 'False'; ExternalVisible := 'False'; ExternalWritable := 'False'} : Bool;
      Ok { ExternalAccessible := 'False'; ExternalVisible := 'False'; ExternalWritable := 'False'} : Bool;
      Nok { ExternalAccessible := 'False'; ExternalVisible := 'False'; ExternalWritable := 'False'} : Bool;
      BtnManConfirmVisible { ExternalAccessible := 'False'; ExternalVisible := 'False'; ExternalWritable := 'False'} : Word;
      BtnManConfirmGreen { ExternalAccessible := 'False'; ExternalVisible := 'False'; ExternalWritable := 'False'} : Word;
      BtnManForceVisible { ExternalAccessible := 'False'; ExternalVisible := 'False'; ExternalWritable := 'False'} : Word;
      BtnManForceGreen { ExternalAccessible := 'False'; ExternalVisible := 'False'; ExternalWritable := 'False'} : Word;
   END_VAR
   VAR_TEMP
      TempNotUsedBool : Bool;
   END_VAR
   VAR CONSTANT
      CMD_TRACK : DWord := 4001;
      OFF : Word := 2#0000000000000000;
      ENABLE : Word := 2#0000000000000001;
      VISIBLE : Word := 2#0000000000000010;
      COLOUR_GREY : Word := 2#0000000000010000;
      COLOUR_WHITE : Word := 2#0000000000100000;
      COLOUR_GREEN : Word := 2#0000000001000000;
      COLOUR_RED : Word := 2#0000000010000000;
      COLOUR_BLUE_FLASH : Word := 2#0000000100000000;
   END_VAR
   VAR_TEMP   // added for the SCL form of the ladder/FBD networks
      _w1 : Bool;
   END_VAR
BEGIN

REGION Network 1: **** 4.4 - Machine status - Input from HMI - Buttons
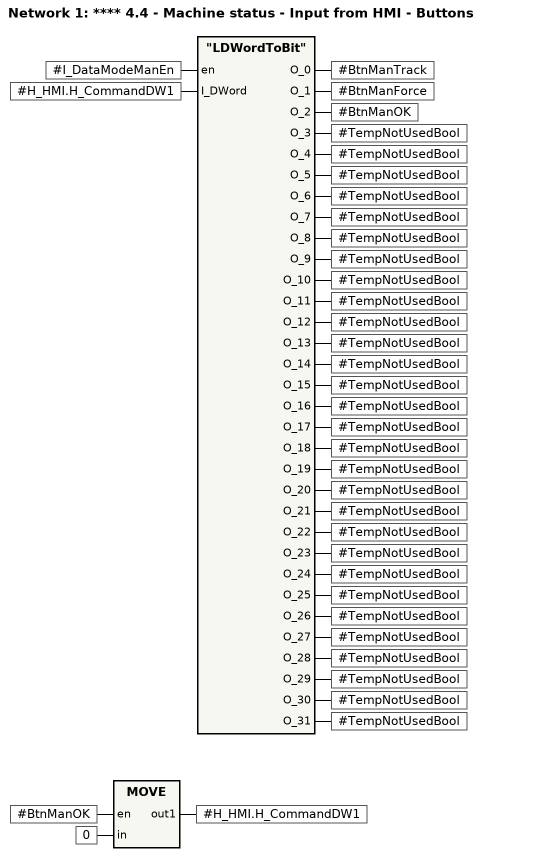
   IF #I_DataModeManEn THEN
       "LDWordToBit"(I_DWord := #H_HMI.H_CommandDW1,
                     O_0 => #BtnManTrack,
                     O_1 => #BtnManForce,
                     O_2 => #BtnManOK,
                     O_3 => #TempNotUsedBool,
                     O_4 => #TempNotUsedBool,
                     O_5 => #TempNotUsedBool,
                     O_6 => #TempNotUsedBool,
                     O_7 => #TempNotUsedBool,
                     O_8 => #TempNotUsedBool,
                     O_9 => #TempNotUsedBool,
                     O_10 => #TempNotUsedBool,
                     O_11 => #TempNotUsedBool,
                     O_12 => #TempNotUsedBool,
                     O_13 => #TempNotUsedBool,
                     O_14 => #TempNotUsedBool,
                     O_15 => #TempNotUsedBool,
                     O_16 => #TempNotUsedBool,
                     O_17 => #TempNotUsedBool,
                     O_18 => #TempNotUsedBool,
                     O_19 => #TempNotUsedBool,
                     O_20 => #TempNotUsedBool,
                     O_21 => #TempNotUsedBool,
                     O_22 => #TempNotUsedBool,
                     O_23 => #TempNotUsedBool,
                     O_24 => #TempNotUsedBool,
                     O_25 => #TempNotUsedBool,
                     O_26 => #TempNotUsedBool,
                     O_27 => #TempNotUsedBool,
                     O_28 => #TempNotUsedBool,
                     O_29 => #TempNotUsedBool,
                     O_30 => #TempNotUsedBool,
                     O_31 => #TempNotUsedBool);
   END_IF;
   IF #BtnManOK THEN #H_HMI.H_CommandDW1 := 0; END_IF;
END_REGION

REGION Network 2: *** 4.4 - Machine status - Calculated *** / **** 4.4 - Machine status - Calculated *** Begin request
   // Start request memory
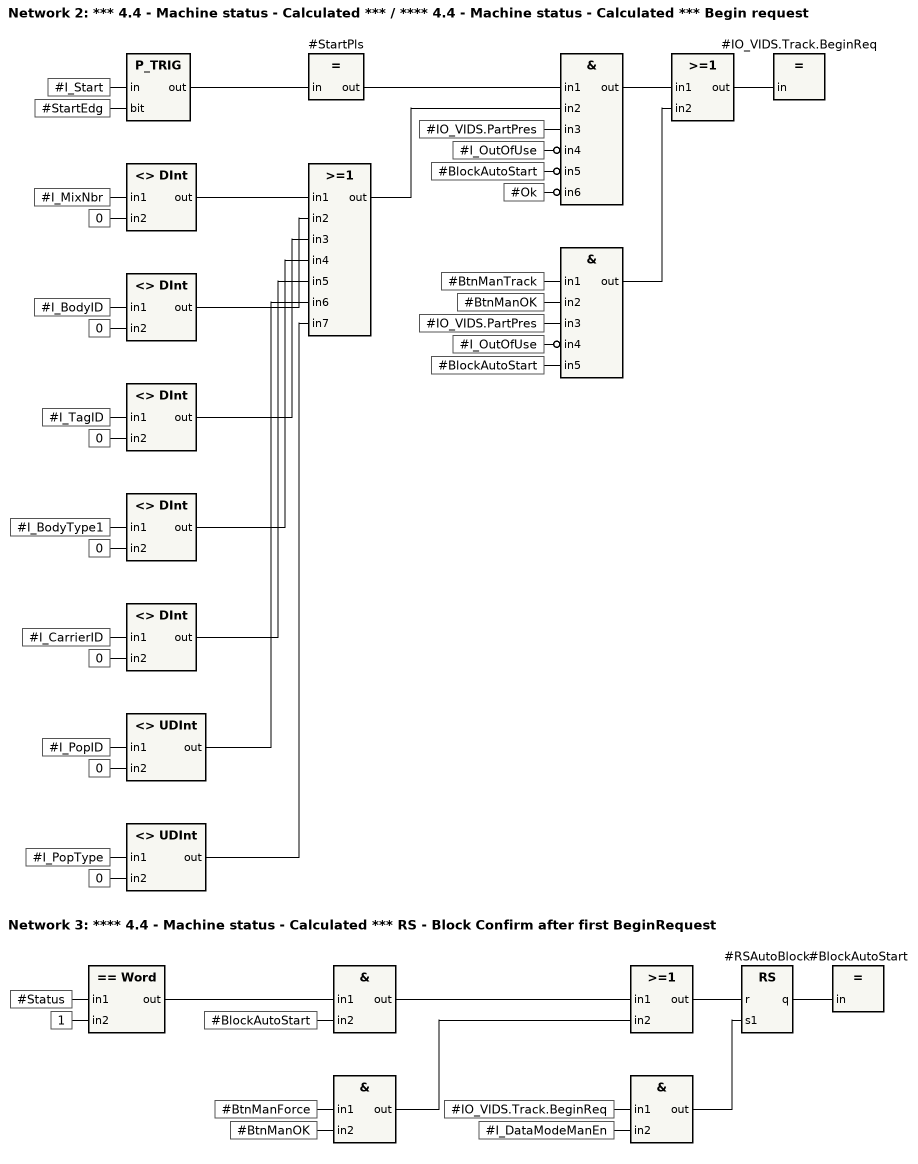
   #_w1 := #I_Start AND NOT #StartEdg;   // rising edge
   #StartEdg := #I_Start;
   #StartPls := #_w1;
   #IO_VIDS.Track.BeginReq := (#_w1 AND ((#I_MixNbr <> 0) OR (#I_BodyID <> 0) OR (#I_TagID <> 0) OR (#I_BodyType1 <> 0) OR (#I_CarrierID <> 0) OR (#I_PopID <> 0) OR (#I_PopType <> 0)) AND #IO_VIDS.PartPres AND NOT #I_OutOfUse AND NOT #BlockAutoStart AND NOT #Ok) OR (#BtnManTrack AND #BtnManOK AND #IO_VIDS.PartPres AND NOT #I_OutOfUse AND #BlockAutoStart);
END_REGION

REGION Network 3: **** 4.4 - Machine status - Calculated *** RS - Block Confirm after first BeginRequest
   IF ((#Status = 1) AND #BlockAutoStart) OR (#BtnManForce AND #BtnManOK) THEN
       #RSAutoBlock := FALSE;   // RS flip-flop
   END_IF;
   IF #IO_VIDS.Track.BeginReq AND #I_DataModeManEn THEN #RSAutoBlock := TRUE; END_IF;
   #BlockAutoStart := #RSAutoBlock;
END_REGION

REGION Network 4: **** 4.4 - Machine status - Calculated *** Memorize parameters
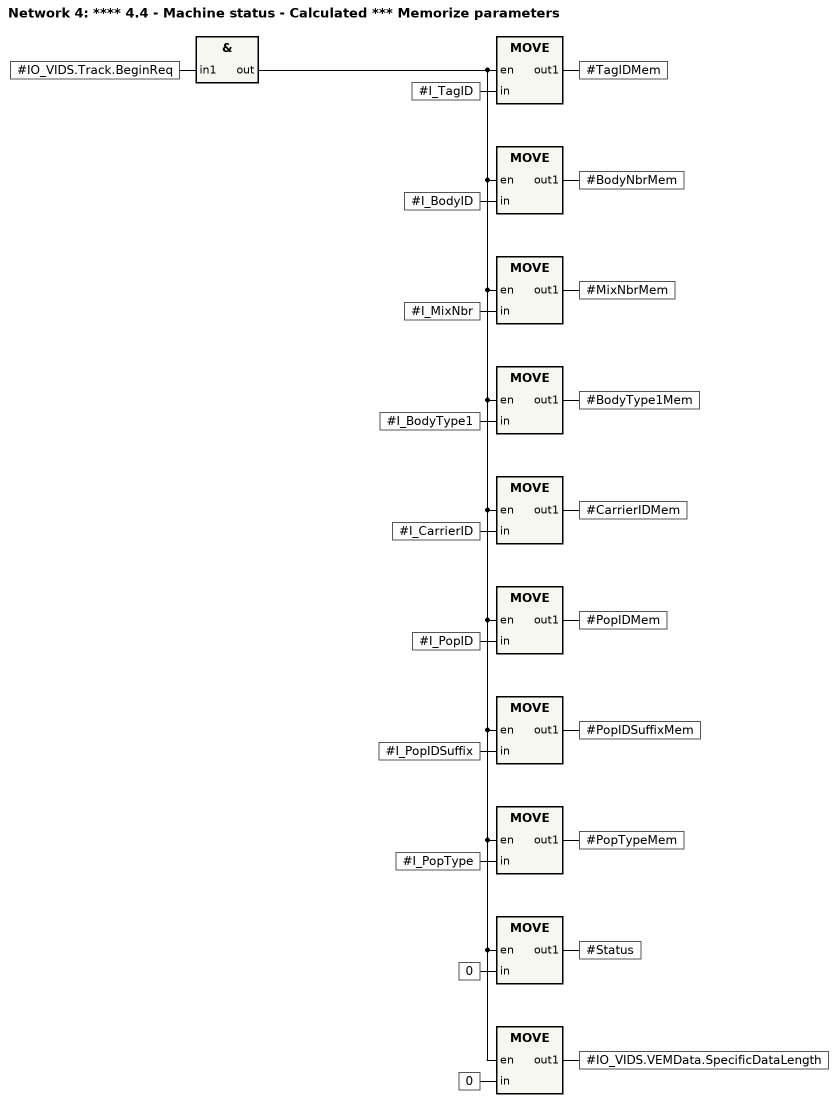
   IF #IO_VIDS.Track.BeginReq THEN
       #TagIDMem := #I_TagID;
       #BodyNbrMem := #I_BodyID;
       #MixNbrMem := #I_MixNbr;
       #BodyType1Mem := #I_BodyType1;
       #CarrierIDMem := #I_CarrierID;
       #PopIDMem := #I_PopID;
       #PopIDSuffixMem := #I_PopIDSuffix;
       #PopTypeMem := #I_PopType;
       #Status := 0;
       #IO_VIDS.VEMData.SpecificDataLength := 0;
   END_IF;
END_REGION

REGION Network 5: *** 4.4 - Machine status - Calculated *** / **** 4.4 - Machine status - Calculated *** Ok to begin
   // Data mode auto - Begin pulse
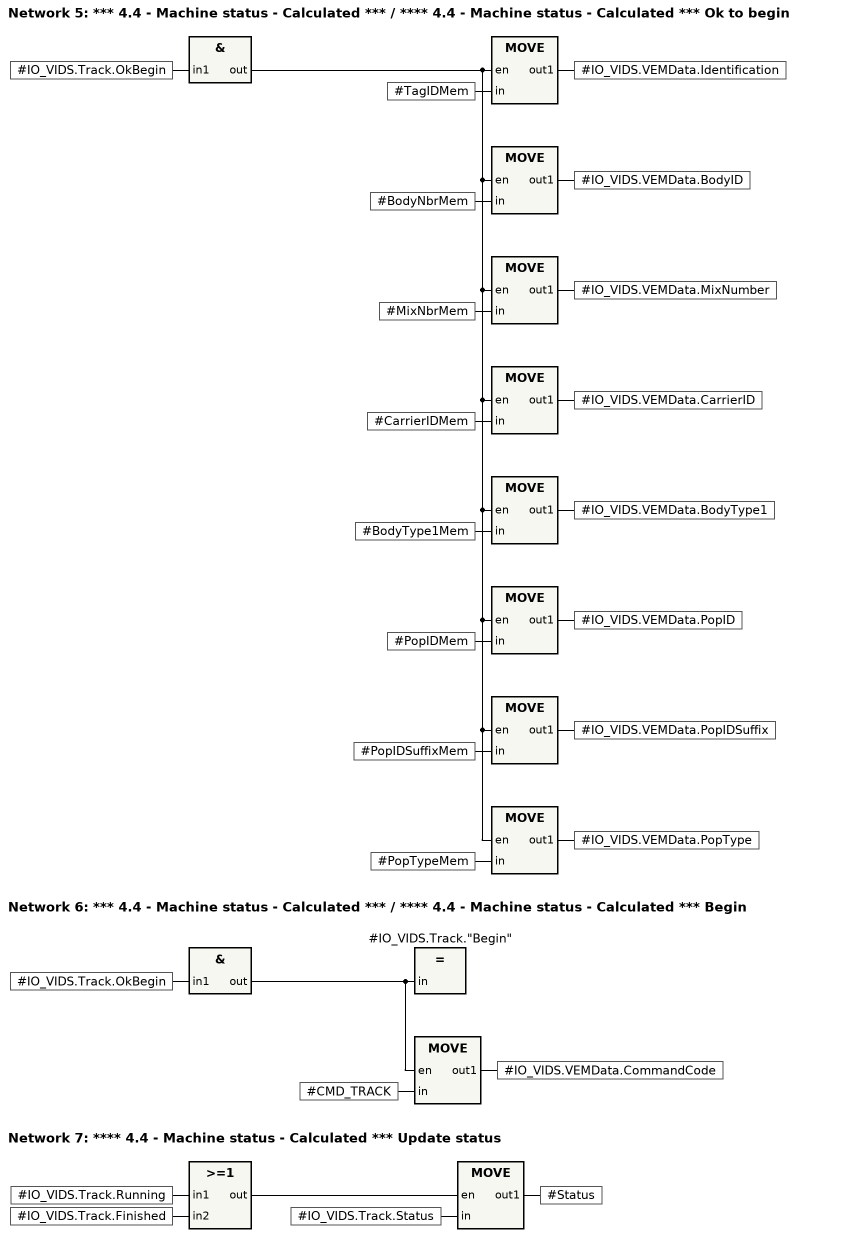
   IF #IO_VIDS.Track.OkBegin THEN
       #IO_VIDS.VEMData.Identification := #TagIDMem;
       #IO_VIDS.VEMData.BodyID := #BodyNbrMem;
       #IO_VIDS.VEMData.MixNumber := #MixNbrMem;
       #IO_VIDS.VEMData.CarrierID := #CarrierIDMem;
       #IO_VIDS.VEMData.BodyType1 := #BodyType1Mem;
       #IO_VIDS.VEMData.PopID := #PopIDMem;
       #IO_VIDS.VEMData.PopIDSuffix := #PopIDSuffixMem;
       #IO_VIDS.VEMData.PopType := #PopTypeMem;
   END_IF;
END_REGION

REGION Network 6: *** 4.4 - Machine status - Calculated *** / **** 4.4 - Machine status - Calculated *** Begin
   // Data mode auto - Begin pulse
   #IO_VIDS.Track."Begin" := #IO_VIDS.Track.OkBegin;
   IF #IO_VIDS.Track.OkBegin THEN #IO_VIDS.VEMData.CommandCode := #CMD_TRACK; END_IF;
END_REGION

REGION Network 7: **** 4.4 - Machine status - Calculated *** Update status
   IF #IO_VIDS.Track.Running OR #IO_VIDS.Track.Finished THEN #Status := #IO_VIDS.Track.Status; END_IF;
END_REGION

REGION Network 8: *** 8 - Outputs *** / **** 4.4 - Machine status - Calculated *** Finished, OK
   // Feedback to process - Tracking finished
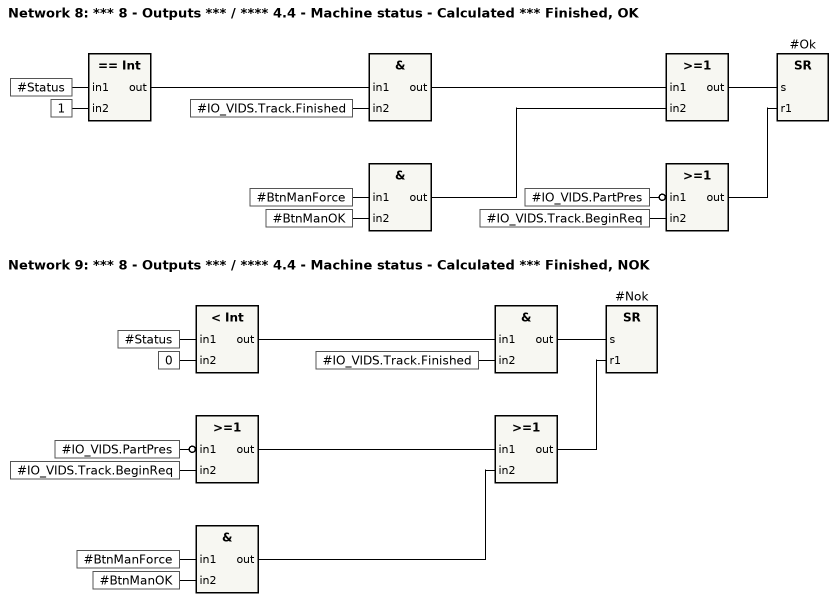
   IF ((#Status = 1) AND #IO_VIDS.Track.Finished) OR (#BtnManForce AND #BtnManOK) THEN
       #Ok := TRUE;   // SR flip-flop
   END_IF;
   IF NOT #IO_VIDS.PartPres OR #IO_VIDS.Track.BeginReq THEN #Ok := FALSE; END_IF;
END_REGION

REGION Network 9: *** 8 - Outputs *** / **** 4.4 - Machine status - Calculated *** Finished, NOK
   // Feedback to process - Tracking finished
   IF (#Status < 0) AND #IO_VIDS.Track.Finished THEN
       #Nok := TRUE;   // SR flip-flop
   END_IF;
   IF NOT #IO_VIDS.PartPres OR #IO_VIDS.Track.BeginReq OR (#BtnManForce AND #BtnManOK) THEN
       #Nok := FALSE;
   END_IF;
END_REGION

REGION Network 10: **** 4.6 - Machine status - Indication *** To HMI - Reset HMI parameters
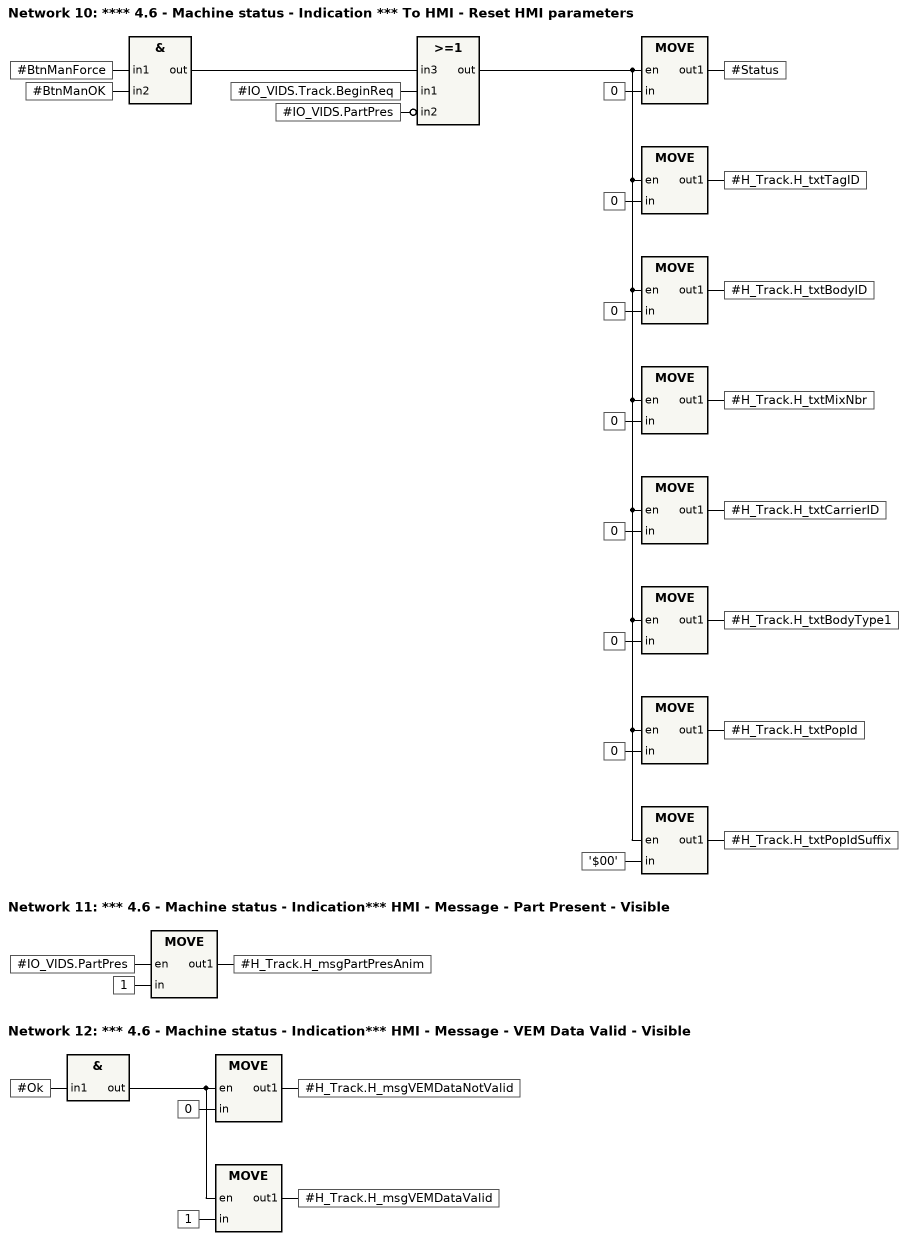
   IF (#BtnManForce AND #BtnManOK) OR #IO_VIDS.Track.BeginReq OR NOT #IO_VIDS.PartPres THEN
       #Status := 0;
       #H_Track.H_txtTagID := 0;
       #H_Track.H_txtBodyID := 0;
       #H_Track.H_txtMixNbr := 0;
       #H_Track.H_txtCarrierID := 0;
       #H_Track.H_txtBodyType1 := 0;
       #H_Track.H_txtPopId := 0;
       #H_Track.H_txtPopIdSuffix := '$00';
   END_IF;
END_REGION

REGION Network 11: *** 4.6 - Machine status - Indication*** HMI - Message - Part Present - Visible
   IF #IO_VIDS.PartPres THEN #H_Track.H_msgPartPresAnim := 1; END_IF;
END_REGION

REGION Network 12: *** 4.6 - Machine status - Indication*** HMI - Message - VEM Data Valid - Visible
   IF #Ok THEN
       #H_Track.H_msgVEMDataNotValid := 0;
       #H_Track.H_msgVEMDataValid := 1;
   END_IF;
END_REGION

REGION Network 13: *** 4.6 - Machine status - Indication*** HMI - Message - VEM Data Not Valid - Visible
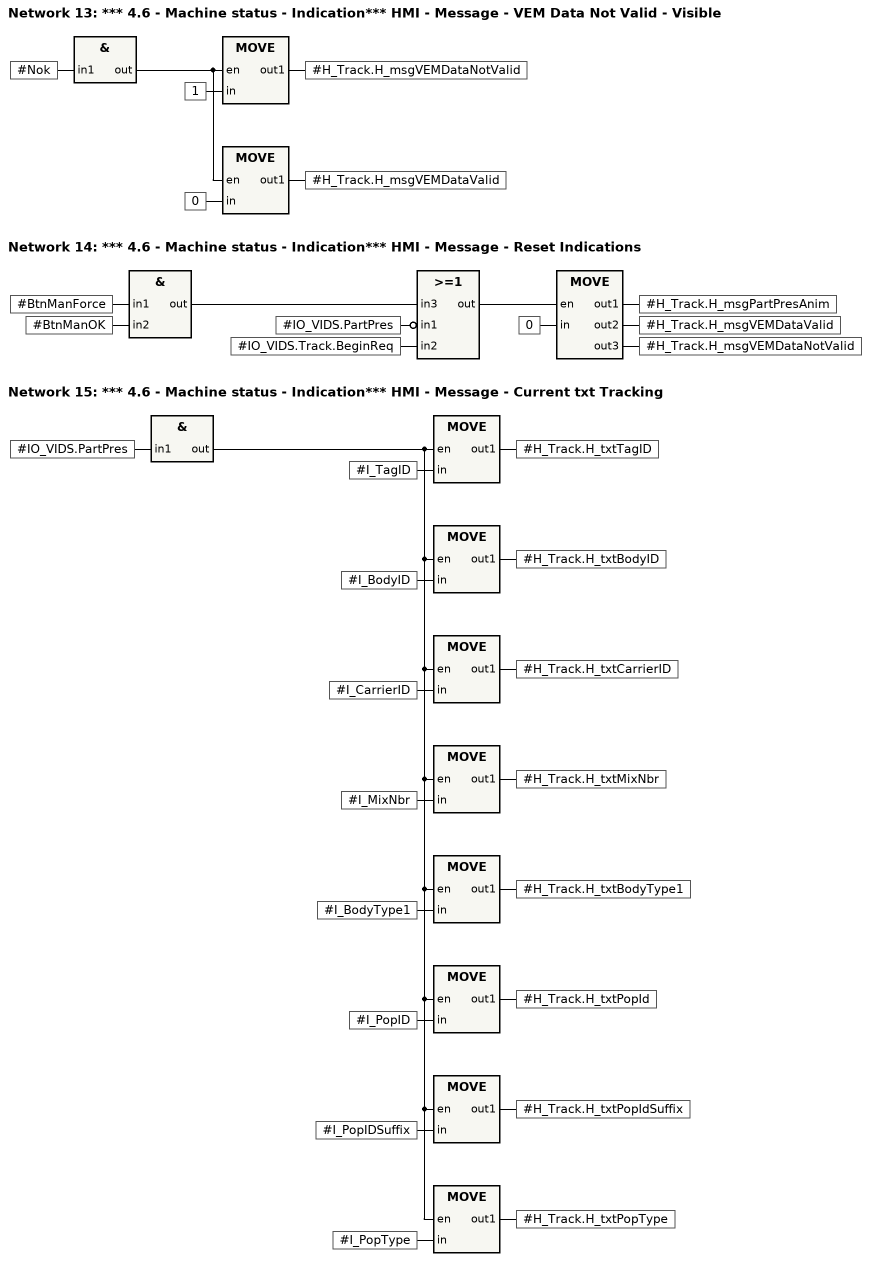
   IF #Nok THEN
       #H_Track.H_msgVEMDataNotValid := 1;
       #H_Track.H_msgVEMDataValid := 0;
   END_IF;
END_REGION

REGION Network 14: *** 4.6 - Machine status - Indication*** HMI - Message - Reset Indications
   IF (#BtnManForce AND #BtnManOK) OR NOT #IO_VIDS.PartPres OR #IO_VIDS.Track.BeginReq THEN
       #H_Track.H_msgPartPresAnim := 0;
       #H_Track.H_msgVEMDataValid := 0;
       #H_Track.H_msgVEMDataNotValid := 0;
   END_IF;
END_REGION

REGION Network 15: *** 4.6 - Machine status - Indication*** HMI - Message - Current txt Tracking
   IF #IO_VIDS.PartPres THEN
       #H_Track.H_txtTagID := #I_TagID;
       #H_Track.H_txtBodyID := #I_BodyID;
       #H_Track.H_txtCarrierID := #I_CarrierID;
       #H_Track.H_txtMixNbr := #I_MixNbr;
       #H_Track.H_txtBodyType1 := #I_BodyType1;
       #H_Track.H_txtPopId := #I_PopID;
       #H_Track.H_txtPopIdSuffix := #I_PopIDSuffix;
       #H_Track.H_txtPopType := #I_PopType;
   END_IF;
END_REGION

REGION Network 16: *** 4.6 - Machine status - Indication*** HMI - Message - Current txt Tracking Reset
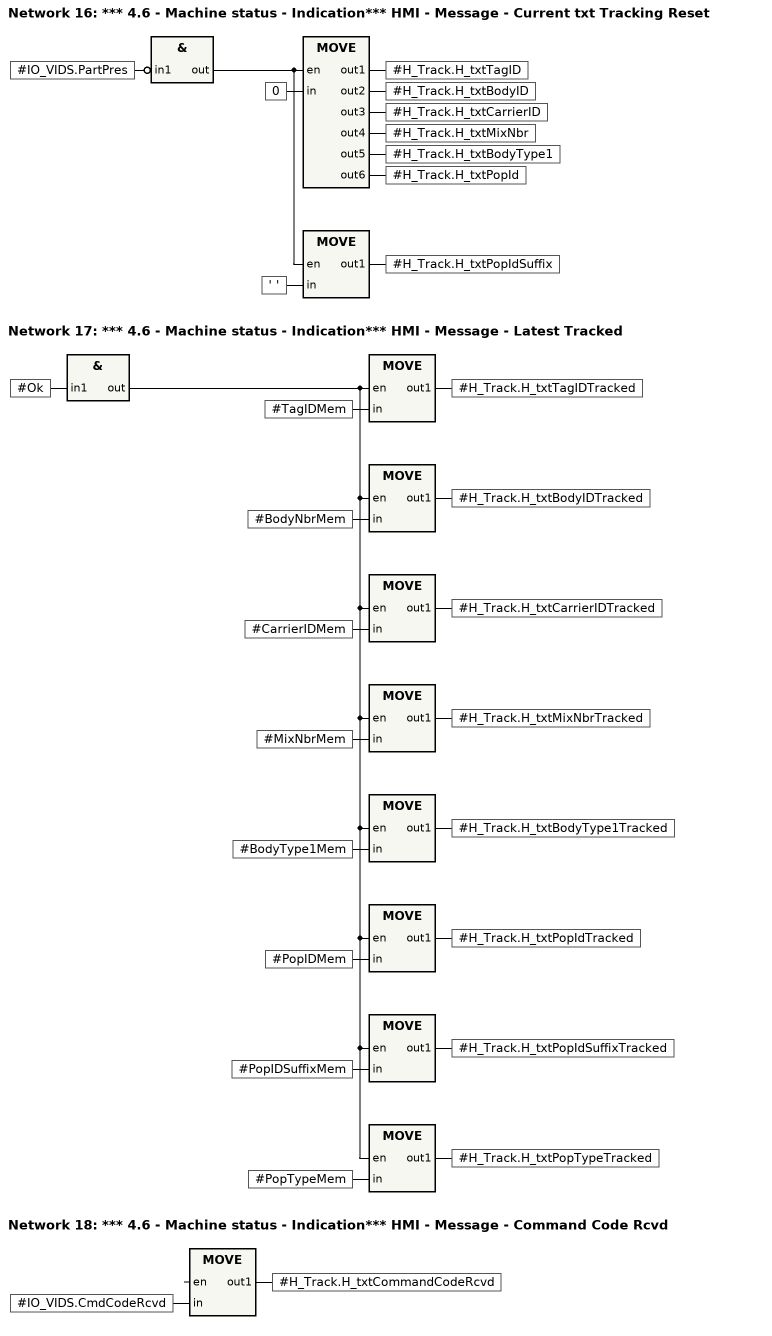
   IF NOT #IO_VIDS.PartPres THEN
       #H_Track.H_txtTagID := 0;
       #H_Track.H_txtBodyID := 0;
       #H_Track.H_txtCarrierID := 0;
       #H_Track.H_txtMixNbr := 0;
       #H_Track.H_txtBodyType1 := 0;
       #H_Track.H_txtPopId := 0;
       #H_Track.H_txtPopIdSuffix := ' ';
   END_IF;
END_REGION

REGION Network 17: *** 4.6 - Machine status - Indication*** HMI - Message - Latest Tracked
   IF #Ok THEN
       #H_Track.H_txtTagIDTracked := #TagIDMem;
       #H_Track.H_txtBodyIDTracked := #BodyNbrMem;
       #H_Track.H_txtCarrierIDTracked := #CarrierIDMem;
       #H_Track.H_txtMixNbrTracked := #MixNbrMem;
       #H_Track.H_txtBodyType1Tracked := #BodyType1Mem;
       #H_Track.H_txtPopIdTracked := #PopIDMem;
       #H_Track.H_txtPopIdSuffixTracked := #PopIDSuffixMem;
       #H_Track.H_txtPopTypeTracked := #PopTypeMem;
   END_IF;
END_REGION

REGION Network 18: *** 4.6 - Machine status - Indication*** HMI - Message - Command Code Rcvd
   #H_Track.H_txtCommandCodeRcvd := #IO_VIDS.CmdCodeRcvd;
END_REGION

REGION Network 19: *** 4.6 - Machine status - Indication*** HMI - Message - Command Code Sent
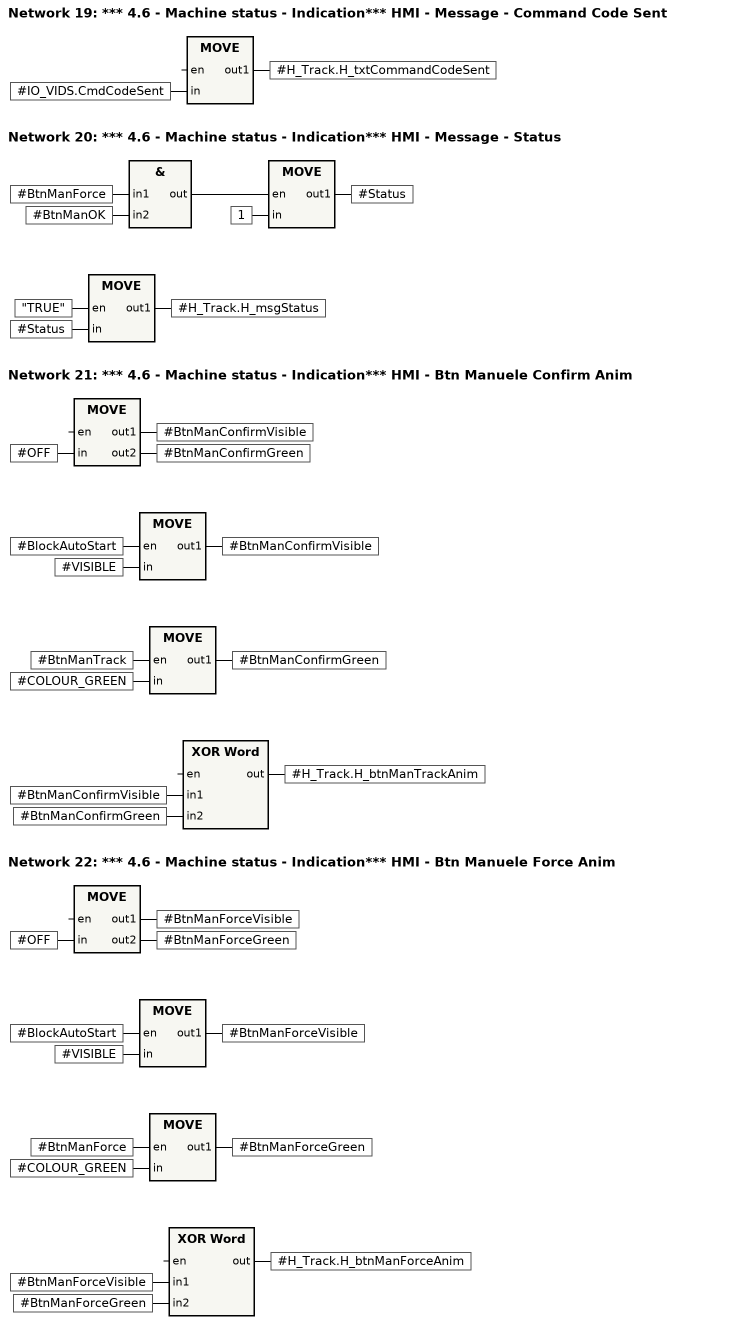
   #H_Track.H_txtCommandCodeSent := #IO_VIDS.CmdCodeSent;
END_REGION

REGION Network 20: *** 4.6 - Machine status - Indication*** HMI - Message - Status
   IF #BtnManForce AND #BtnManOK THEN #Status := 1; END_IF;
   IF "TRUE" THEN #H_Track.H_msgStatus := #Status; END_IF;
END_REGION

REGION Network 21: *** 4.6 - Machine status - Indication*** HMI - Btn Manuele Confirm Anim
   #BtnManConfirmVisible := #OFF;
   #BtnManConfirmGreen := #OFF;
   IF #BlockAutoStart THEN #BtnManConfirmVisible := #VISIBLE; END_IF;
   IF #BtnManTrack THEN #BtnManConfirmGreen := #COLOUR_GREEN; END_IF;
   #H_Track.H_btnManTrackAnim := #BtnManConfirmVisible XOR #BtnManConfirmGreen;
END_REGION

REGION Network 22: *** 4.6 - Machine status - Indication*** HMI - Btn Manuele Force Anim
   #BtnManForceVisible := #OFF;
   #BtnManForceGreen := #OFF;
   IF #BlockAutoStart THEN #BtnManForceVisible := #VISIBLE; END_IF;
   IF #BtnManForce THEN #BtnManForceGreen := #COLOUR_GREEN; END_IF;
   #H_Track.H_btnManForceAnim := #BtnManForceVisible XOR #BtnManForceGreen;
END_REGION

REGION Network 23: *** 4.6 - Machine status - Indication*** HMI - Btn Manuele Confirm Anim
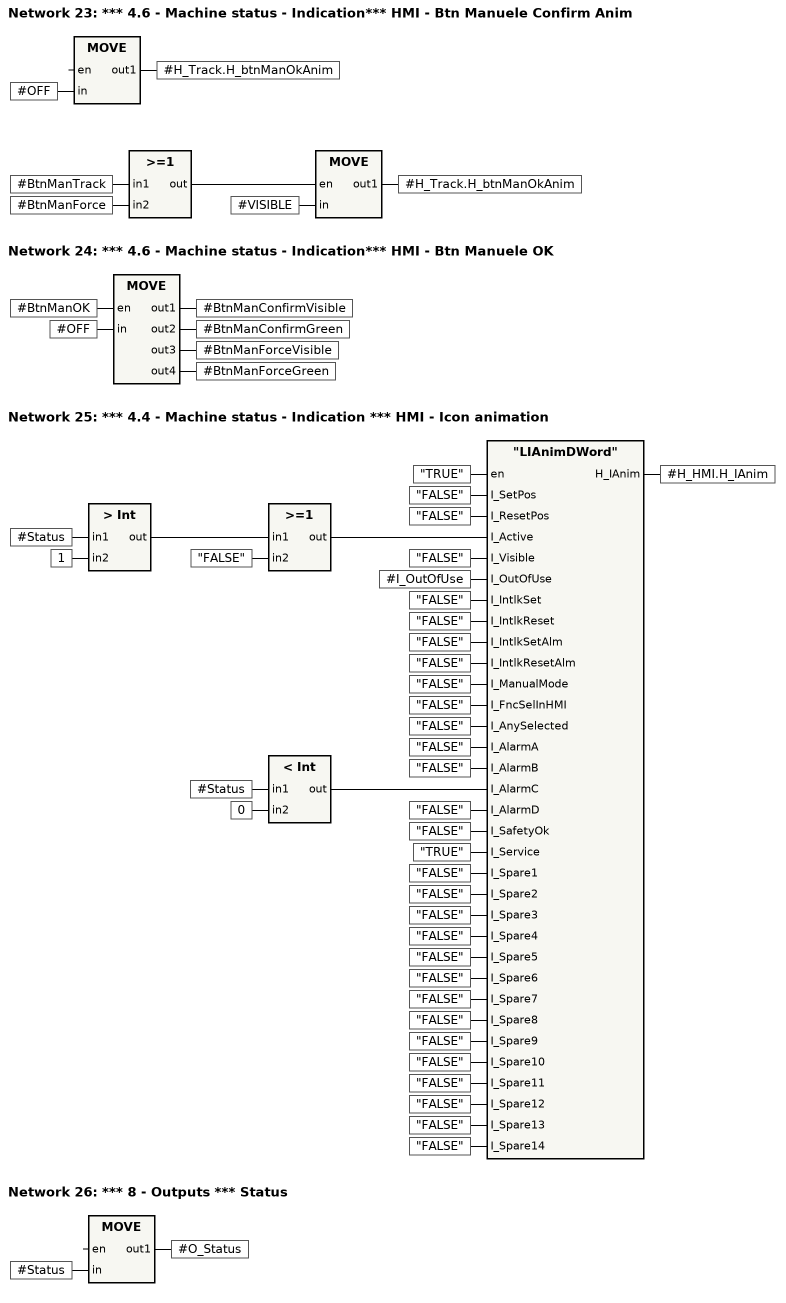
   #H_Track.H_btnManOkAnim := #OFF;
   IF #BtnManTrack OR #BtnManForce THEN #H_Track.H_btnManOkAnim := #VISIBLE; END_IF;
END_REGION

REGION Network 24: *** 4.6 - Machine status - Indication*** HMI - Btn Manuele OK
   IF #BtnManOK THEN
       #BtnManConfirmVisible := #OFF;
       #BtnManConfirmGreen := #OFF;
       #BtnManForceVisible := #OFF;
       #BtnManForceGreen := #OFF;
   END_IF;
END_REGION

REGION Network 25: *** 4.4 - Machine status - Indication *** HMI - Icon animation
   IF "TRUE" THEN
       "LIAnimDWord"(I_SetPos := "FALSE",
                     I_ResetPos := "FALSE",
                     I_Active := (#Status > 1) OR "FALSE",
                     I_Visible := "FALSE",
                     I_OutOfUse := #I_OutOfUse,
                     I_IntlkSet := "FALSE",
                     I_IntlkReset := "FALSE",
                     I_IntlkSetAlm := "FALSE",
                     I_IntlkResetAlm := "FALSE",
                     I_ManualMode := "FALSE",
                     I_FncSelInHMI := "FALSE",
                     I_AnySelected := "FALSE",
                     I_AlarmA := "FALSE",
                     I_AlarmB := "FALSE",
                     I_AlarmC := #Status < 0,
                     I_AlarmD := "FALSE",
                     I_SafetyOk := "FALSE",
                     I_Service := "TRUE",
                     I_Spare1 := "FALSE",
                     I_Spare2 := "FALSE",
                     I_Spare3 := "FALSE",
                     I_Spare4 := "FALSE",
                     I_Spare5 := "FALSE",
                     I_Spare6 := "FALSE",
                     I_Spare7 := "FALSE",
                     I_Spare8 := "FALSE",
                     I_Spare9 := "FALSE",
                     I_Spare10 := "FALSE",
                     I_Spare11 := "FALSE",
                     I_Spare12 := "FALSE",
                     I_Spare13 := "FALSE",
                     I_Spare14 := "FALSE",
                     H_IAnim => #H_HMI.H_IAnim);
   END_IF;
END_REGION

